# B&R Automation Studio project WithUpgradesWorking23_08_24
Automation Studio 4.9

## Configuration Config1

CPU X90CP174.48-00, AutomationRuntime I4.93, Build 4.1.2, Safety 0.0, Vc V4.72.6

### Hardware
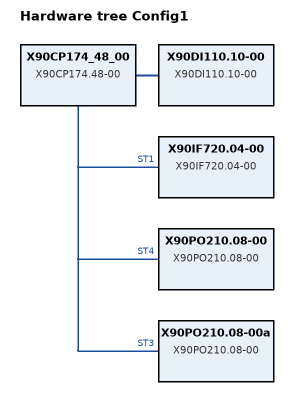
```
X90CP174_48_00 : X90CP174.48-00 v1.4.5.0  [X1 -> X1.SL]
  Module X1 (Type=X1, Virtual=true, Version=1.4.5.0)
    Connection (Connector=SL, TargetModule=X90CP174_48_00, TargetConnector=X1)
    ChannelConfig01 = 42
    DigitalFilterPin01 = 200
    ChannelConfig02 = 42
    DigitalFilterPin02 = 200
    ChannelConfig03 = 42
    DigitalFilterPin03 = 200
    ChannelConfig04 = 42
    DigitalFilterPin04 = 200
    ChannelConfig05 = 42
    DigitalFilterPin05 = 200
    ChannelConfig06 = 42
    DigitalFilterPin06 = 200
    ChannelConfig07 = 42
    DigitalFilterPin07 = 200
    ChannelConfig08 = 42
    DigitalFilterPin08 = 200
    ChannelConfig12 = 81
    ChannelConfig13 = 72
    DigitalFilterPin13 = 200
    ChannelConfig17 = 80
    ChannelConfig18 = 80
    ChannelConfig19 = 80
    ChannelConfig20 = 80
    ChannelConfig21 = 80
    ChannelConfig22 = 80
    ChannelConfig23 = 80
    IN2_InputFilter_Pin23 = 3
    ChannelConfig24 = 80
    ChannelConfig27 = 1
    ChannelConfig28 = 41
    DigitalFilterPin28 = 200
    ChannelConfig37 = 1
    LoadType37 = 2
    ChannelConfig38 = 1
    LoadType38 = 2
    ChannelConfig39 = 1
    ChannelConfig41 = 1
    LoadType41 = 2
    ChannelConfig42 = 1
    ChannelConfig45 = 1
    LoadType45 = 2
    ChannelConfig46 = 1
    LoadType46 = 2
    core = core1
  Connector IF2:
    ActivateDevice = 1
    Mode = Manual
    InternetAddress = 169.254.143.70
    SubnetMask = 255.255.0.0
    InaNodeNumber = 0
    ActivateSnmp = 2
  Connector IF3:
    DNAConfiguration = manual
    CycleTime = 1000
  ConfigurationID = Project_Config1
  UserPartitionSize = 0
  VolatileGlobalPvSize = 100000000
  IdleTaskClass = 5
  TaskClassIdleTime = 5000
  CyclicTaskClassCount = 6
  Cyclic1Duration = 1000
  Cyclic1Tolerance = 10000
  Cyclic2Duration = 4000
  Cyclic2Tolerance = 20000
  Cyclic3Duration = 10000
  Cyclic3Tolerance = 20000
  Cyclic4Duration = 20000
  Cyclic4Tolerance = 20000
  Cyclic5Duration = 50000
  Cyclic5Tolerance = 50000
  Cyclic6Duration = 100000
  Cyclic6Tolerance = 100000
  Cyclic7Duration = 100000
  Cyclic7Tolerance = 1000000
  Cyclic8Duration = 10000
  Cyclic8Tolerance = 30000000
  FileDevice1
  FileDeviceName1 = C
  FileDevicePath1 = C:/vikings/missions
  FileDevice2
  FileDeviceName2 = plc
  FileDevicePath2 = USER_PATH
  FtpUser1
  FtpUsername1 = viking  // viking
  FtpUserPassword1 = Dom8yxQRfEJkQNN0YFGST8fEunO7EPE9T/2DWtETr4U=  // viking
  FtpUserSalt1 = iKbGjPE0
  FTPAccessRight1 = 0
  ActivateOpcUa = 1
  OpcUaInformationModels_PV_Version = 1
X90DI110.10-00 : X90DI110.10-00 v1.1.1.0  [ST -> X90CP174_48_00.ST2]
  Mode_DigIn01 = 22k_pnp
  InputFilter01 = 200
  Mode_DigIn02 = 22k_pnp
  InputFilter02 = 200
  Mode_DigIn03 = 22k_pnp
  InputFilter03 = 200
  Mode_DigIn04 = 22k_pnp
  Mode_DigIn05 = 22k_pnp
  Mode_DigIn06 = 22k_pnp
  Mode_DigIn07 = 22k_pnp
  InputFilter07 = 200
  Mode_DigIn08 = 22k_pnp
  Mode_DigIn09 = 22k_pnp
  InputFilter09 = 200
  Mode_DigIn10 = 22k_pnp
  InputFilter10 = 200
X90IF720.04-00 : X90IF720.04-00 v1.0.2.0  [ST -> X90CP174_48_00.ST1]
  Connector IF4:
    Baudrate = 115200
X90PO210.08-00 : X90PO210.08-00 v1.4.0.0  [ST -> X90CP174_48_00.ST4]
X90PO210.08-00a : X90PO210.08-00 v1.4.0.0  [ST -> X90CP174_48_00.ST3]
```

### IoMap.iom - X90CP174_48_00/IoMap.iom
```iecst
VAR_CONFIG
	::gCooling.outputs.do_fan[1] AT %QX."X1".DigitalOutput46;
	::gCooling.inputs.ai_coolingTemp[0] AT %IW."X1".AnalogInput17;
	::gCooling.inputs.ai_coolingTemp[1] AT %IW."X1".AnalogInput19;
	::gCooling.outputs.do_pump[1] AT %QX."X1".DigitalOutput45;
	::gCooling.outputs.do_fan[0] AT %QX."X1".DigitalOutput37;
	::gCooling.outputs.do_pump[0] AT %QX."X1".DigitalOutput38;
	::gSafetyChain.inputs.di_interlockWheelFR_OK AT %IX."X1".DigitalInput05;
	::gSafetyChain.inputs.di_shutdownRight_OK AT %IX."X1".DigitalInput07;
	::gSafetyChain.inputs.di_interlockWheelFL_OK AT %IX."X1".DigitalInput06;
	::gSafetyChain.inputs.di_interlockWheelRR_OK AT %IX."X1".DigitalInput08;
	::gSafetyChain.inputs.di_shutdownLeft_OK AT %IX."X1".DigitalInput01;
	::gSafetyChain.inputs.di_shutdownCockpit_OK AT %IX."X1".DigitalInput02;
	::gSafetyChain.inputs.di_inertiaSwitch_OK AT %IX."X1".DigitalInput03;
	::gSafetyChain.inputs.di_BOTS_OK AT %IX."X1".DigitalInput04;
	::gSafetyChain.inputs.di_TSMS_OK AT %IX."X1".DigitalInput13;
	::gSteeringAngle.inputs.angleSensor AT %IW."X1".AnalogInput20;
	::gTorqueSensor.inputs.torque2 AT %IW."X1".AnalogInput21;
	::gBraking.inputs.ai_brakePressureFront AT %IW."X1".AnalogInput22;
	::gTorqueSensor.inputs.torque1 AT %IW."X1".AnalogInput24;
	::gBraking.inputs.ai_brakePressureRear AT %IW."X1".AnalogInput18;
	::gInverters.inverter[0].inputs.di_deratingActive AT %IX."X90DI110.10-00".DigitalInput06;
	::gInverters.inverter[1].inputs.di_deratingActive AT %IX."X90DI110.10-00".DigitalInput04;
	::gInverters.inverter[2].inputs.di_deratingActive AT %IX."X90DI110.10-00".DigitalInput08;
	::gInverters.inverter[3].inputs.di_deratingActive AT %IX."X90DI110.10-00".DigitalInput05;
	::gInverters.inverter[0].outputs.do_enable AT %QX."X90PO210.08-00a".DigitalOutput01;
	::gInverters.inverter[1].outputs.do_enable AT %QX."X90PO210.08-00a".DigitalOutput07;
	::gInverters.inverter[3].outputs.do_enable AT %QX."X90PO210.08-00a".DigitalOutput06;
	::gInverters.inverter[2].outputs.do_torqueLimitActive AT %QX."X90PO210.08-00a".DigitalOutput02;
	::gInverters.inverter[0].outputs.do_torqueLimitActive AT %QX."X90PO210.08-00a".DigitalOutput03;
	::gInverters.inverter[1].outputs.do_torqueLimitActive AT %QX."X90PO210.08-00a".DigitalOutput08;
	::gInverters.output.do_enableInv34 AT %QX."X90PO210.08-00a".DigitalOutput04;
	::gInverters.inverter[2].outputs.do_enable AT %QX."X90PO210.08-00".DigitalOutput03;
	::gInverters.inverter[3].outputs.do_torqueLimitActive AT %QX."X90PO210.08-00".DigitalOutput02;
	::gInverters.output.do_enableInv12 AT %QX."X90PO210.08-00".DigitalOutput05;
	::gSafetyChain.inputs.di_TS_Container AT %IX."X90DI110.10-00".DigitalInput07;
	::gSafetyChain.inputs.di_interlockWheelRL_OK AT %IX."X90DI110.10-00".DigitalInput10;
	::gSafetyChain.inputs.di_supply AT %IX."X90DI110.10-00".DigitalInput09;
	::gSafetyChain.inputs.di_BSPD_OK AT %IX."X90DI110.10-00".DigitalInput03;
	::gSafetyChain.inputs.di_interlockHVD_OK AT %IX."X90DI110.10-00".DigitalInput01;
	::gSafetyChain.inputs.di_interlockTSMP_OK AT %IX."X90DI110.10-00".DigitalInput02;
	::gRTDS.outputs.do_RTDS AT %QX."X1".DigitalOutput41;
	::gBraking.outputs.do_brakeLight AT %QX."X1".DigitalOutput42;
	gRTDS.inputs.im_RTDS_Current AT %IW."X1".Current41;
	::gCooling.inputs.im_pumpCurrent[1] AT %IW."X1".Current45;
	::gCooling.inputs.im_pumpCurrent[0] AT %IW."X1".Current38;
	::gInverters.output.do_powerInv12 AT %QX."X1".DigitalOutput39;
	::gInverters.output.do_powerInv34 AT %QX."X1".DigitalOutput27;
	::gLowVoltageBattery.inputs.ai_voltage AT %IW."X1".AnalogInput12;
	::gLowVoltageBattery.inputs.ai_current AT %IW."X1".AnalogInput23;
	::gSafetyChain.inputs.di_interlockMotorRL_OK AT %IX."X1".DigitalInput28;
END_VAR
```

## Logical view

Binary libraries used (declarations not repeated): operator, runtime, astime, AsIecCon, standard, AsIODiag, brsystem, asstring, ArCan, brdkUSB, AsIO, AsBrStr, sys_lib, FileIO, AsUSB, DataObj, brdkSTR, NcGlobal, MTTypes, dvframe, MpAlarmX, MpBase, MpRecipe, MpData, MTFilter 5.24.1

### Global.typ - Global data types
```iecst
TYPE
	CAN_STATES :
		(
		S_INIT,
		S_INIT_TX,
		S_INIT_RX,
		S_RUNNING,
		S_ERROR,
		S_IDLE
		);
END_TYPE
```

### Package Logical/Libraries - Global libraries

### Library Logical/Libraries/brdkSIM (ANSIC)

#### Types.typ
```iecst
TYPE
	brdkSIM_status_typ : 	STRUCT
		fbStatus : brdkSIM_STATUS_typ;
		error : BOOL;
		errorCode : UINT;
	END_STRUCT;
	brdkSIM_STATUS_typ :
		(
		brdkSIM_NOT_ENABLED := 0,
		brdkSIM_BUSY := 10,
		brdkSIM_RUNNING := 20,
		brdkSIM_ERROR := 200
		);
	brdkSimInput_internal_typ : 	STRUCT
		state : USINT;
		AsIOEnableForcing_0 : AsIOEnableForcing;
		AsIOSetForceValue_0 : AsIOSetForceValue;
		AsIODisableForcing_0 : AsIODisableForcing;
		oldSetValue : UDINT;
	END_STRUCT;
	brdkSimOutput_internal_typ : 	STRUCT
		state : USINT;
		pvStatus : UINT;
		pvAdr : UDINT;
		pvLen : UDINT;
		pvCheck : UINT;
		pvCmpString : STRING[4];
		boolVar : BOOL;
	END_STRUCT;
END_TYPE
```

#### brdkSimInput.c
```c
#include <bur/plctypes.h>
#include <AsIO.h>
#include <AsBrStr.h>

#ifdef __cplusplus
	extern "C"
	{
#endif
	#include "brdkSIM.h"
#ifdef __cplusplus
	};
#endif

#define false 0
#define true 1

/* TODO: Add your comment here */
void brdkSimInput(struct brdkSimInput* inst)
{
	int i;

	if (!inst->enable && inst->internal.state > 0 && inst->internal.state < 50) {
		inst->internal.state = 50;
	}

	switch (inst->internal.state) {
		case 0: //wait for enable force
			inst->status.fbStatus = brdkSIM_NOT_ENABLED;
			inst->status.error = false;
			inst->status.errorCode = 0;
			inst->internal.oldSetValue = 0;
			if (inst->enable) {
				inst->internal.state = 10;
			}
			break;

		case 10: //enable force
			inst->status.fbStatus = brdkSIM_BUSY;
			if (!inst->internal.AsIOEnableForcing_0.enable) {
				inst->internal.AsIOEnableForcing_0.enable = true;
				inst->internal.AsIOEnableForcing_0.pDatapoint = (UDINT)&inst->dpName;		// set pointer to the var name (address)
				inst->internal.state = 20;
			}
			break;

		case 20: //wait for AsIOEnableForcing_0 fb to be ready
			if (inst->internal.AsIOEnableForcing_0.status == ERR_OK) {
				inst->internal.AsIOEnableForcing_0.enable = false;					// remember to set enable false so the fb is ready for the next dp
				AsIOEnableForcing(&inst->internal.AsIOEnableForcing_0);
				inst->internal.state = 30;
			}
			else if (inst->internal.AsIOEnableForcing_0.status != ERR_OK && inst->internal.AsIOEnableForcing_0.status != ERR_FUB_BUSY && inst->internal.AsIOEnableForcing_0.status != ERR_FUB_ENABLE_FALSE) {
				inst->status.fbStatus = brdkSIM_ERROR;
				inst->status.error = true;
				inst->status.errorCode = inst->internal.AsIOEnableForcing_0.status;
				inst->internal.state = 200;
			}
			break;

		case 30: //AsIOSetForceValue_0 fb use to control force value
			inst->status.fbStatus = brdkSIM_RUNNING;
			inst->internal.AsIOSetForceValue_0.enable 		= true;
			inst->internal.AsIOSetForceValue_0.pDatapoint	= (UDINT)&inst->dpName;		// set pointer to the dp name (address)
			inst->internal.AsIOSetForceValue_0.value 		= inst->setValue;						// set the force value

			if (inst->internal.AsIOSetForceValue_0.status != ERR_OK && inst->internal.AsIOSetForceValue_0.status != ERR_FUB_BUSY && inst->internal.AsIOSetForceValue_0.status != ERR_FUB_ENABLE_FALSE) {
				inst->status.fbStatus = brdkSIM_ERROR;
				inst->status.error = true;
				inst->status.errorCode = inst->internal.AsIOSetForceValue_0.status;
				inst->internal.state = 200;
			}
			break;

		case 50: //set value to 0 before disable
			inst->status.fbStatus = brdkSIM_BUSY;
			if (inst->internal.AsIOSetForceValue_0.value != 0) {
				inst->internal.AsIOSetForceValue_0.enable 		= true;
				inst->internal.AsIOSetForceValue_0.pDatapoint	= (UDINT)&inst->dpName;		// set pointer to the dp name (address)
				inst->internal.AsIOSetForceValue_0.value 		= 0;									// set the force value
				inst->internal.oldSetValue 						= 0;

				if (inst->internal.AsIOSetForceValue_0.status != ERR_OK && inst->internal.AsIOSetForceValue_0.status != ERR_FUB_BUSY && inst->internal.AsIOSetForceValue_0.status != ERR_FUB_ENABLE_FALSE) {
					inst->status.fbStatus = brdkSIM_ERROR;
					inst->status.error = true;
					inst->status.errorCode = inst->internal.AsIOSetForceValue_0.status;
					inst->internal.state = 200;
				}
				else {
					inst->internal.state 	= 60;
				}
			}
			else {
				inst->internal.state 	= 60;
			}
			break;

		case 60: //wait for AsIODisableForcing_0 fb to be ready
			inst->internal.AsIOSetForceValue_0.enable 		= false;
			inst->internal.AsIODisableForcing_0.enable 		= true;
			inst->internal.AsIODisableForcing_0.pDatapoint 	= (UDINT)&inst->dpName;		// set pointer to the dp name (address)
			AsIODisableForcing(&inst->internal.AsIODisableForcing_0);

			if (inst->internal.AsIODisableForcing_0.status == ERR_OK) {
				inst->internal.AsIODisableForcing_0.enable 	= false;						// remember to set enable false so the fb is ready for the next dp
				inst->internal.state = 0;
			}
			else if (inst->internal.AsIODisableForcing_0.status != ERR_OK && inst->internal.AsIODisableForcing_0.status != ERR_FUB_BUSY && inst->internal.AsIODisableForcing_0.status != ERR_FUB_ENABLE_FALSE) {
				inst->status.fbStatus = brdkSIM_ERROR;
				inst->status.error = true;
				inst->status.errorCode = inst->internal.AsIODisableForcing_0.status;
				inst->internal.state = 200;
			}
			break;

		case 200: //error
			inst->internal.AsIOEnableForcing_0.enable = false;
			inst->internal.AsIOSetForceValue_0.enable = false;
			inst->internal.AsIODisableForcing_0.enable 	= false;
			inst->internal.oldSetValue = 0;

			if (!inst->enable) {
				inst->status.error = false;
				inst->status.errorCode = 0;
				inst->internal.state 	= 0;
			}
	}

	AsIOEnableForcing(&inst->internal.AsIOEnableForcing_0);
	AsIOSetForceValue(&inst->internal.AsIOSetForceValue_0);
	AsIODisableForcing(&inst->internal.AsIODisableForcing_0);
}
```

#### brdkSimOutput.c
```c
#include <bur/plctypes.h>
#include <sys_lib.h>
#include <AsBrStr.h>

#ifdef __cplusplus
	extern "C"
	{
#endif
	#include "brdkSIM.h"
#ifdef __cplusplus
	};
#endif

#define false 0
#define true 1

/* TODO: Add your comment here */
void brdkSimOutput(struct brdkSimOutput* inst)
{
	if (!inst->enable && inst->internal.state > 0) {
		inst->internal.state = 0;
		inst->internal.pvAdr = 0;
		inst->internal.pvCheck = 0;
		inst->internal.pvLen = 0;
		inst->internal.pvStatus = 0;
		inst->internal.state = 0;
	}

	switch (inst->internal.state) {
		case 0: //wait for enable
			inst->status.fbStatus = brdkSIM_NOT_ENABLED;
			inst->status.error = false;
			inst->status.errorCode = 0;

			if(inst->enable) {
				brsstrcpy((UDINT)inst->internal.pvCmpString, (UDINT) "");
				inst->internal.pvCheck = brsstrcmp((UDINT)inst->pvName, (UDINT)inst->internal.pvCmpString);
				if(inst->internal.pvCheck != 0) {
					inst->internal.state = 10;
				}
				else {
					inst->status.fbStatus = brdkSIM_ERROR;
					inst->status.error = true;
					inst->status.errorCode = 1000;
					inst->internal.state = 200;
				}
			}
			break;

		case 10: //get address of the pv
			inst->status.fbStatus = brdkSIM_BUSY;
			inst->internal.pvStatus = PV_xgetadr((UDINT)&inst->pvName, (UDINT)&inst->internal.pvAdr, (UDINT)&inst->internal.pvLen);

			if(inst->internal.pvStatus != 0) {
				inst->status.fbStatus = brdkSIM_ERROR;
				inst->status.error = true;
				inst->status.errorCode = inst->internal.pvStatus;
				inst->internal.state = 200;
			}
			else {
				inst->internal.state = 20;
			}
			break;

		case 20: //check value
			inst->status.fbStatus = brdkSIM_RUNNING;
			brsmemcpy((UDINT)&inst->actValue, (UDINT)inst->internal.pvAdr, inst->internal.pvLen);
			break;

		case 200: //error
			break;
	}
}
```

### Library Logical/Libraries/sduVikings (IEC)

#### calculateSensorNetOut.st
```iecst
(* TODO: Add your comment here *)
FUNCTION_BLOCK calculateSensorNetOut
//	y = a1 + a2*x^1 + a3*x^2 + a4*x^3 + ... + a8*x^7
	y := polyCoeffs[0];
	FOR i := 1 TO 8 DO
		// y = y + a^i
		y := y + polyCoeffs[i] * EXPT(INT_TO_REAL(input), i);
	END_FOR;
	output := y;
END_FUNCTION_BLOCK
```

### globalEventLog.typ - Global data types
```iecst
TYPE
	gEventLog_typ : 	STRUCT
		newEventString : STRING[80];
		logNewEvent : BOOL;
		eventIndex : UINT := 0;
		events : ARRAY[0..EVENT_LOG_LENGTH]OF STRING[80];
		resetEventLog : BOOL;
	END_STRUCT;
END_TYPE
```

### globalEventLog.var - Global variables
```iecst
VAR CONSTANT
	EVENT_LOG_LENGTH : UINT := 100;
END_VAR
VAR
	gEventLog : gEventLog_typ;
END_VAR
```

### globalStateMachine.typ
```iecst
TYPE
	gStateMachine_cmd_typ : 	STRUCT
		forceIO : BOOL;
		changeMission : BOOL;
		loadMission : BOOL;
		saveMission : BOOL;
	END_STRUCT;
	gStateMachine_data_typ : 	STRUCT
		dummy : USINT;
	END_STRUCT;
	gStateMachine_inputs_typ : 	STRUCT
		dummy : INT;
	END_STRUCT;
	gStateMachine_outputs_typ : 	STRUCT
		dummy : USINT;
	END_STRUCT;
	gStateMachine_status_typ : 	STRUCT
		readyForStateDrive : BOOL;
		stateNameOld : STRING[80];
		stateName : STRING[80];
		stateChangeAllowed : BOOL;
		stateOld : states_typ;
		state : states_typ;
		instruction : STRING[80];
		instructionIndex : instructionIndex;
		mission : STRING[80];
		missionIndex : missionIndex_typ;
		stateChangeTimeout : BOOL;
	END_STRUCT;
	gStateMachine_typ : 	STRUCT
		status : gStateMachine_status_typ;
		outputs : gStateMachine_outputs_typ;
		data : gStateMachine_data_typ;
		cmd : gStateMachine_cmd_typ;
		inputs : gStateMachine_inputs_typ;
	END_STRUCT;
	instructionIndex :
		(
		INST_INITIALIZING,
		INST_PRESS_SAFETY_BUTTON,
		INST_SC_NOT_ENABLED,
		INST_PRESS_TRACTIVE_BUTTON,
		INST_AMS_NOT_READY,
		INST_PRESS_BRAKE,
		INST_TORQUE_PEDAL_FAULT,
		INST_PRE_CHARGING,
		INST_PRESS_DRIVE_BUTTON,
		INST_FIX_ERROR,
		INST_CLOSE_SAFETY_CHAIN,
		INST_IN_DRIVE
		);
	states_typ :
		(
		STATE_INITIALIZE,
		STATE_IDLE,
		STATE_ENABLING_SC,
		STATE_SC_ENABLED,
		STATE_PRECHARGING,
		STATE_TRACTIVE,
		STATE_DRIVE,
		STATE_ERROR
		);
END_TYPE
```

### globalStateMachine.var
```iecst
VAR
	gStateMachine : gStateMachine_typ;
END_VAR
```

### Program Logical/SM/StateMachine (IEC)

#### Types.typ - Local data types
```iecst
TYPE
	this_typ : 	STRUCT
		TON_initialization : TON;
		instructionList : ARRAY[0..25]OF STRING[80];
	END_STRUCT;
END_TYPE
```

#### stateInit.st
```iecst
(* State Initialize *)
ACTION stateInit:

	this.TON_initialization();

	(* Start timer *)
	IF NOT this.TON_initialization.IN THEN
		this.TON_initialization.IN := TRUE;
	END_IF

END_ACTION

(* Conditions for state change for STATE_INITIALIZE*)
ACTION stateChangeInit:

	(* Initialization done change state to ready *)
	IF this.TON_initialization.Q THEN
		this.TON_initialization.IN := FALSE;
		gStateMachine.status.state := STATE_IDLE;
	END_IF

END_ACTION
```

#### stateEnablingSC.st
```iecst
(* State Ready *)
ACTION stateEnablingSC:
	(* Update instruction string *)
	gStateMachine.status.instructionIndex := INST_SC_NOT_ENABLED;
END_ACTION

(* Conditions for state change for STATE_ENABLE_SAFETY_CHAIN *)
ACTION stateChangeEnablingSC:
	IF gStateMachine.status.stateChangeAllowed THEN
		(* If message received from AMS saying that SC is enabled *)
		IF gAMS.status.scEnabled THEN
			gStateMachine.status.state := STATE_SC_ENABLED;
		END_IF

		(* If safety chain is broken go to state 'stateError' *)
		IF NOT gSafetyChain.status.scOK_notEnabled THEN
			gStateMachine.status.state 	:= STATE_ERROR;
			gAMS.cmd.abort 				:= TRUE;
		END_IF

		IF gStateMachine.status.stateChangeTimeout THEN
			gAMS.cmd.abort := TRUE;
			gStateMachine.status.state 			    := STATE_IDLE;
		END_IF;
	END_IF;

END_ACTION
```

#### logEvent.st
```iecst
ACTION logEvent:

	gEventLog.events[gEventLog.eventIndex] := gEventLog.newEventString;

	gEventLog.eventIndex 				   := gEventLog.eventIndex + 1;
	IF gEventLog.eventIndex > EVENT_LOG_LENGTH THEN
		gEventLog.eventIndex := 0;
	END_IF;

	gEventLog.events[gEventLog.eventIndex] := '';

END_ACTION

ACTION resetEventLog:

	FOR gEventLog.eventIndex := 0 TO EVENT_LOG_LENGTH DO
		gEventLog.events[gEventLog.eventIndex] := '';
	END_FOR;
	gEventLog.eventIndex := 0;

END_ACTION
```

#### forceIO.st
```iecst
ACTION initForceIO:
	brdkSimInput_0[0].dpName  := '%IX.X1.DigitalInput05'; 			//::gSafetyChain.inputs.di_interlockWheelFR_OK
	brdkSimInput_0[1].dpName  := '%IX.X1.DigitalInput07'; 			//:gSafetyChain.inputs.di_shutdownRight_OK
	brdkSimInput_0[2].dpName  := '%IX.X1.DigitalInput06'; 			//::gSafetyChain.inputs.di_interlockWheelFL_OK
	brdkSimInput_0[3].dpName  := '%IX.X1.DigitalInput08'; 			//::gSafetyChain.inputs.di_interlockWheelRR_OK
	brdkSimInput_0[4].dpName  := '%IX.X1.DigitalInput01'; 			//::gSafetyChain.inputs.di_shutdownLeft_OK
	brdkSimInput_0[5].dpName  := '%IX.X1.DigitalInput02'; 			//::gSafetyChain.inputs.di_shutdownCockpit_OK
	brdkSimInput_0[6].dpName  := '%IX.X1.DigitalInput03'; 			//::gSafetyChain.inputs.di_inertiaSwitch_OK
	brdkSimInput_0[7].dpName  := '%IX.X1.DigitalInput04'; 			//::gSafetyChain.inputs.di_BOTS_OK
	brdkSimInput_0[8].dpName  := '%IX.X1.DigitalInput13'; 			//::gSafetyChain.inputs.di_TSMS_OK
	brdkSimInput_0[9].dpName  := '%IW.X1.AnalogInput20'; 			//::gSteeringAngle.inputs.angleSensor
	brdkSimInput_0[10].dpName := '%IW.X1.AnalogInput21'; 			//::gTorqueSensor.inputs.torque2
	brdkSimInput_0[11].dpName := '%IW.X1.AnalogInput22'; 			//::gBraking.inputs.ai_brakePressureFront
	brdkSimInput_0[12].dpName := '%IW.X1.AnalogInput24'; 			//::gTorqueSensor.inputs.torque1
	brdkSimInput_0[13].dpName := '%IW.X1.AnalogInput18'; 			//::gBraking.inputs.ai_brakePressureRear
	brdkSimInput_0[14].dpName := '%IX.IF6.ST2.DigitalInput07'; //::gSafetyChain.inputs.di_TS_Container
	brdkSimInput_0[15].dpName := '%IX.IF6.ST2.DigitalInput10'; //::gSafetyChain.inputs.di_interlockWheelRL_OK
	brdkSimInput_0[16].dpName := '%IX.IF6.ST2.DigitalInput09'; //::gSafetyChain.inputs.di_supply
	brdkSimInput_0[17].dpName := '%IX.IF6.ST2.DigitalInput03'; //::gSafetyChain.inputs.di_BSPD_OK
	brdkSimInput_0[18].dpName := '%IX.IF6.ST2.DigitalInput01'; //::gSafetyChain.inputs.di_interlockHVD_OK
	brdkSimInput_0[19].dpName := '%IX.IF6.ST2.DigitalInput02'; //::gSafetyChain.inputs.di_interlockTSMP_OK
END_ACTION

ACTION forceIO:

	FOR i := 0 TO SIM_INPUTS-1 DO
		brdkSimInput_0[i].enable := gStateMachine.cmd.forceIO;
	END_FOR;

	brdkSimInput_0[0].setValue  := gSafetyChain.cmd.di_interlockWheelFR_OK;
	brdkSimInput_0[1].setValue  := gSafetyChain.cmd.di_shutdownRight_OK;
	brdkSimInput_0[2].setValue  := gSafetyChain.cmd.di_interlockWheelFL_OK;
	brdkSimInput_0[3].setValue  := gSafetyChain.cmd.di_interlockWheelRR_OK;
	brdkSimInput_0[4].setValue  := gSafetyChain.cmd.di_shutdownLeft_OK;
	brdkSimInput_0[5].setValue  := gSafetyChain.cmd.di_shutdownCockpit_OK;
	brdkSimInput_0[6].setValue  := gSafetyChain.cmd.di_inertiaSwitch_OK;
	brdkSimInput_0[7].setValue  := gSafetyChain.cmd.di_BOTS_OK;
	brdkSimInput_0[8].setValue  := gSafetyChain.cmd.di_TSMS_OK;
	brdkSimInput_0[9].setValue  := gSteeringAngle.cmd.angleSensor;
	brdkSimInput_0[10].setValue := gTorqueSensor.cmd.torque2;
	brdkSimInput_0[11].setValue := gBraking.cmd.brakePressureFront;
	brdkSimInput_0[12].setValue := gTorqueSensor.cmd.torque1;
	brdkSimInput_0[13].setValue := gBraking.cmd.brakePressureRear;
	brdkSimInput_0[14].setValue := gSafetyChain.cmd.di_TS_Container;
	brdkSimInput_0[15].setValue := gSafetyChain.cmd.di_interlockWheelRL_OK;
	brdkSimInput_0[16].setValue := gSafetyChain.cmd.di_supply;
	brdkSimInput_0[17].setValue := gSafetyChain.cmd.di_BSPD_OK;
	brdkSimInput_0[18].setValue := gSafetyChain.cmd.di_interlockHVD_OK;
	brdkSimInput_0[19].setValue := gSafetyChain.cmd.di_interlockTSMP_OK;

	FOR i := 0 TO SIM_INPUTS-1 DO
		brdkSimInput_0[i]();
	END_FOR;

END_ACTION
```

#### changeStateDelay.st
```iecst
//
ACTION changeStateDelay:
	IF gStateMachine.status.state <> STATE_TRACTIVE THEN
		gStateMachine.status.readyForStateDrive := FALSE;
	END_IF

	TON_stateChange(IN := gStateMachine.status.stateOld <> gStateMachine.status.state);
	IF TON_stateChange.Q THEN
		gStateMachine.status.stateOld := gStateMachine.status.state;
	END_IF;

	gStateMachine.status.stateChangeAllowed := gStateMachine.status.stateOld = gStateMachine.status.state;

END_ACTION
```

### Variables.var
```iecst
VAR
	TON_persistancetimer : TON;
	i : USINT;
END_VAR
```

### globalInverters.typ
```iecst
TYPE
	gInverters_typ : 	STRUCT
		data : gInverters_data_typ;
		cmd : gInverters_cmd_typ;
		status : gInverters_status_typ;
		output : gInverters_output_typ;
		inverter : ARRAY[0..3]OF gInverters_inverter_typ;
	END_STRUCT;
	gInverters_data_typ : 	STRUCT
		powerLimitKW : REAL;
		powerLimit : REAL;
		averageVelocityKmh : REAL;
		deratingStatic : REAL;
		acceleration_0to100kmh_inSecs : TIME;
		negativeTorqueLimGain : REAL;
		torqueSetpointGain : REAL;
		MaxSpeedRPM : REAL;
		powerLimitMargin : REAL;
		powerLimitKwInverter : ARRAY[0..3]OF REAL;
		powerBias : ARRAY[0..3]OF REAL;
		rearBias : REAL;
	END_STRUCT;
	gInverters_cmd_typ : 	STRUCT
		enableRegenerativeBraking : BOOL;
		enableTractionControl : BOOL;
		enablePowerLimiter : BOOL;
		enableTorqueVectoring : BOOL;
		enableTorqueLimiter : BOOL;
		enableFrontRearDistribution : BOOL;
		enableMotorPairShutdown : BOOL;
		powerCycle : BOOL;
		exitDrive : BOOL;
		manualControl : BOOL;
		enableConfigurationDuringDrive : BOOL; (*True = All inverter control parameters are enabled to be changed during drive*)
		autoReset : BOOL;
		stopInverters : BOOL;
		activateInverters : BOOL;
		powerCyclePair12 : BOOL;
		powerCyclePair34 : BOOL;
	END_STRUCT;
	gInverters_output_typ : 	STRUCT
		do_enableInv34 : BOOL; (*BA1*)
		do_enableInv12 : BOOL; (*BA1*)
		do_powerInv12 : BOOL;
		do_powerInv34 : BOOL;
	END_STRUCT;
	gInverters_status_typ : 	STRUCT
		deratingStaticPercent : REAL;
		configurationEnabled : BOOL;
		errorCanFramesLost : ARRAY[0..1]OF BOOL;
		regenerativeBrakingAvailable : BOOL;
		torqueBasedThrottle : BOOL;
	END_STRUCT;
	gInverters_inverter_typ : 	STRUCT
		status : gInverters_inverter_status_typ;
		outputs : gInverters_inverter_outputs_typ;
		data : gInverters_inverter_data_typ;
		inputs : gInverters_inverter_inputs_typ;
		cmd : gInverters_inverter_cmd_typ;
	END_STRUCT;
	gInverters_inverter_status_typ : 	STRUCT
		ok : BOOL;
		substate : USINT;
		stateName : STRING[80];
		state : gInverterStates;
		returnState : gInverterStates; (*State to return back to if an error occurs here*)
		errorTimeout : BOOL;
		inverterEnabled : BOOL;
		unknownMessageReceived : BOOL;
		unknownMessageID : UDINT;
		inverterDisconnected : BOOL;
		locationName : STRING[80];
		location : INVERTER_LOCATIONS_TYP;
		deratingLaunchProfilePercent : REAL;
		deratingPowerLimiterPercent : REAL;
		deratingFrontRearDistribution : REAL;
		deratingTorqueVectoringPercent : REAL;
		deratingTotalPercent : REAL;
	END_STRUCT;
	gInverters_inverter_data_typ : 	STRUCT
		torqueOutput : REAL;
		torqueOutputPercent : REAL;
		tempMotor : REAL;
		tempInverter : REAL;
		tempIGBT : REAL;
		actualVelocityKmh : REAL;
		actualVelocity : REAL;
		torqueCurrent : REAL;
		torqueMagnitizingCurrent : REAL;
		speedDerating : REAL;
		maxSpeed : REAL; (*Max speed recorded in last run, remember to implement in code*)
		TON_errorTimer : TON; (*Timer to monitor how long an inverter has been in the error state*)
		regenerativeBraking : REAL;
		regenerativeBrakingPercent : REAL;
	END_STRUCT;
	gInverters_inverter_inputs_typ : 	STRUCT
		com_systemReady : BOOL;
		com_error : BOOL;
		com_warning : BOOL;
		com_quitDcOn : BOOL;
		com_dcOn : BOOL;
		com_quitInverterOn : BOOL;
		com_inverterOn : BOOL;
		com_derating : BOOL;
		com_actualVelocity : INT;
		com_torqueCurrent : INT;
		com_magnetizingCurrent : INT;
		com_tempMotor : INT;
		com_tempInverter : INT;
		com_tempIGBT : INT;
		com_errorDiagnostics : UDINT;
		di_deratingActive : BOOL;
	END_STRUCT;
	gInverters_inverter_cmd_typ : 	STRUCT
		enableInverter : BOOL;
		stopInverter : BOOL;
		startInverter : BOOL;
		shutdownByPartner : BOOL;
		powerCycle : BOOL;
	END_STRUCT;
	gInverters_inverter_outputs_typ : 	STRUCT
		torqueEnable : BOOL;
		do_torqueLimitActive : BOOL; (*BE2*)
		do_enable : BOOL; (*BE1*)
		com_errorReset : BOOL;
		com_enable : BOOL;
		com_dcOn : BOOL;
		com_interverOn : BOOL;
		com_targetVelocity : INT;
		com_targetTorque : INT;
		com_torqueLimitPos : INT;
		com_torqueLimitNeg : INT;
	END_STRUCT;
	missionIndex_typ :
		(
		MISSION_NONE,
		MISSION_ACCELERATION,
		MISSION_SKIDPAD,
		MISSION_SPRINT,
		MISSION_ENDURANCE,
		MISSION_BRAKE_TEST,
		MISSION_TESTING
		);
	INVERTER_LOCATIONS_TYP :
		(
		FL,
		FR,
		RL,
		RR
		);
	gInverterStates :
		(
		INV_STATE_INIT,
		INV_STATE_IDLE,
		INV_STATE_SWITCH_ON,
		INV_STATE_DRIVE,
		INV_STATE_ERROR,
		INV_STATE_SWITCH_OFF,
		INV_STATE_POWER_CYCLE
		);
END_TYPE
```

### globalInverters.var
```iecst
VAR
	gInverters : {REDUND_UNREPLICABLE} gInverters_typ;
	CONVERTER_PEAK_CURRENT : REAL := 105.00;
END_VAR
VAR CONSTANT
	INVERTER_COUNT : USINT := 3;
END_VAR
```

### Program Logical/Inverters/CAN/CAN (IEC)

#### Bus.st
```iecst
ACTION Bus:

	CASE bus[i].communicationState OF
		S_INIT:
			(* PLC is not simulated. It is run on an actual PLC *)
			IF NOT gIsSimulation THEN

				(* Configure CAN port *)
				bus[i].ArCanSetBaudrate_0.DeviceName	:= bus[i].deviceName;

				bus[i].ArCanSetBaudrate_0.Execute 	:= TRUE;
				IF bus[i].ArCanSetBaudrate_0.Done THEN
					bus[i].communicationState := S_INIT_TX;
				END_IF;

				IF bus[i].ArCanSetBaudrate_0.Error THEN
					bus[i].communicationState := S_ERROR;
				END_IF;

			ELSE
				(* PLC is simulated. It is run in the simulator and no hardware is connnected *)
				bus[i].communicationState := S_IDLE;
			END_IF;
		S_INIT_TX:
			(* Configure send function block *)
			bus[i].ArCanSend_0.Enable 		:= TRUE;
			bus[i].ArCanSend_0.DeviceName 	:= bus[i].deviceName;

			IF bus[i].ArCanSend_0.Active THEN
				bus[i].communicationState := S_INIT_RX;
			END_IF;

			IF bus[i].ArCanSend_0.Error THEN
				bus[i].communicationState := S_ERROR;
			END_IF;

		S_INIT_RX:
			(* Configure receive function block *)
			bus[i].ArCanReceive_0.Enable 		:= TRUE;
			bus[i].ArCanReceive_0.DeviceName 	:= bus[i].deviceName;

			IF bus[i].ArCanReceive_0.Active THEN
				(* CAN port successfully enabled *)
				bus[i].communicationState := S_RUNNING;
			END_IF;

			IF bus[i].ArCanReceive_0.Error THEN
				bus[i].communicationState := S_ERROR;
			END_IF

		S_RUNNING:
			(* Send messages *)
			Send_Bus;

			(* Receive messages *)
			Receive_Bus;

		S_ERROR: // Error
			IF bus[i].ArCanSend_0.Error THEN
				bus[i].ArCanSend_0(Enable := FALSE);
				bus[i].ArCanSend_0(Enable := TRUE);
			END_IF;

			IF bus[i].ArCanReceive_0.Error THEN
				bus[i].ArCanReceive_0(Enable := FALSE);
				bus[i].ArCanReceive_0(Enable := TRUE);
			END_IF;

			IF bus[i].ArCanReceive_0.Error = FALSE AND bus[i].ArCanSend_0.Error = FALSE AND bus[i].ArCanSetBaudrate_0.Error = FALSE THEN
				bus[i].communicationState 	:= S_INIT;
			END_IF;
		S_IDLE: // Do nothing
	END_CASE

	IF NOT gIsSimulation THEN
		bus[i].ArCanSetBaudrate_0();
		bus[i].ArCanReceive_0();
		bus[i].ArCanSend_0();
	END_IF;

	// Service disconnection timers
	serviceDisconnectionDetection;

END_ACTION
```

#### receiveMsgs.st
```iecst
(* Inverter 1, Actual value 1 *)
ACTION Inv_ActualValue1:

	gInverters.inverter[inverterId].inputs.com_systemReady 			:= bus[i].ArCanReceive_0.ReceivedFrame.Data[1].0;
	gInverters.inverter[inverterId].inputs.com_error 				:= bus[i].ArCanReceive_0.ReceivedFrame.Data[1].1;
	gInverters.inverter[inverterId].inputs.com_warning 				:= bus[i].ArCanReceive_0.ReceivedFrame.Data[1].2;
	gInverters.inverter[inverterId].inputs.com_quitDcOn 			:= bus[i].ArCanReceive_0.ReceivedFrame.Data[1].3;
	gInverters.inverter[inverterId].inputs.com_dcOn 				:= bus[i].ArCanReceive_0.ReceivedFrame.Data[1].4;
	gInverters.inverter[inverterId].inputs.com_quitInverterOn		:= bus[i].ArCanReceive_0.ReceivedFrame.Data[1].5;
	gInverters.inverter[inverterId].inputs.com_inverterOn 			:= bus[i].ArCanReceive_0.ReceivedFrame.Data[1].6;
	gInverters.inverter[inverterId].inputs.com_derating 			:= bus[i].ArCanReceive_0.ReceivedFrame.Data[1].7;

	memcpy(ADR(gInverters.inverter[inverterId].inputs.com_actualVelocity), 		ADR(bus[i].ArCanReceive_0.ReceivedFrame.Data[2]), 2);
	memcpy(ADR(gInverters.inverter[inverterId].inputs.com_torqueCurrent), 	  	ADR(bus[i].ArCanReceive_0.ReceivedFrame.Data[4]), 2);
	memcpy(ADR(gInverters.inverter[inverterId].inputs.com_magnetizingCurrent), 	ADR(bus[i].ArCanReceive_0.ReceivedFrame.Data[6]), 2);

END_ACTION

(* Inverter 1, Actual value 2 *)
ACTION Inv_ActualValue2:
	memcpy(ADR(gInverters.inverter[inverterId].inputs.com_tempMotor), 			ADR(bus[i].ArCanReceive_0.ReceivedFrame.Data[0]), 2);
	memcpy(ADR(gInverters.inverter[inverterId].inputs.com_tempInverter), 		ADR(bus[i].ArCanReceive_0.ReceivedFrame.Data[2]), 2);
	memcpy(ADR(gInverters.inverter[inverterId].inputs.com_errorDiagnostics),	ADR(bus[i].ArCanReceive_0.ReceivedFrame.Data[4]), 2);
	memcpy(ADR(gInverters.inverter[inverterId].inputs.com_tempIGBT),  			ADR(bus[i].ArCanReceive_0.ReceivedFrame.Data[6]), 2);
END_ACTION
```

#### Send_Bus.st
```iecst
ACTION Send_Bus:

	(* Set timer *)
	bus[i].TON_sendTimer.PT := T#30ms;

	(* If timer runs out *)
	IF bus[i].TON_sendTimer.Q THEN
		// Make sure there is free spots in the TX message buffer
		IF bus[i].ArCanSend_0.NumberOfFreeBuffers > 1010 THEN
			(* Go through each message. Encode and send them *)
			FOR j := 2*i TO (2*i)+1 DO
				(* Set ID of message *)
				bus[i].sendMessages := bus[i].sendMessages + 1;
				CASE j OF
					0: bus[i].ArCanSend_0.Frame.ID := TX_CAN_ID_BASE + 16#084;
					1: bus[i].ArCanSend_0.Frame.ID := TX_CAN_ID_BASE + 16#085;
					2: bus[i].ArCanSend_0.Frame.ID := TX_CAN_ID_BASE + 16#088;
					3: bus[i].ArCanSend_0.Frame.ID := TX_CAN_ID_BASE + 16#089;
					ELSE
				END_CASE
				IF bus[i].ArCanSend_0.Frame.ID <> 0 THEN
					encodeAndSendMessage; // Encode and send message
				END_IF;
			END_FOR;
		END_IF;

		(* Reset timer *)
		bus[i].TON_sendTimer(IN:=FALSE);
	END_IF

	(* Start timer *)
	bus[i].TON_sendTimer(IN:=TRUE);

END_ACTION
```

### Program Logical/Inverters/Control/Control (IEC)

#### Main.st - Init, cyclic, exit code
```iecst
PROGRAM _INIT

	// Initialize inverter locations
	gInverters.inverter[FL].status.location 	:= FL;
	gInverters.inverter[FR].status.location 	:= FR;
	gInverters.inverter[RL].status.location 	:= RL;
	gInverters.inverter[RR].status.location 	:= RR;

	FOR i := 0 TO INVERTER_COUNT DO
		// Initialize inverter location names
		CASE gInverters.inverter[i].status.location OF
			FL: gInverters.inverter[i].status.locationName := 'FL';
			FR: gInverters.inverter[i].status.locationName := 'FR';
			RL: gInverters.inverter[i].status.locationName := 'RL';
			RR: gInverters.inverter[i].status.locationName := 'RR';
		END_CASE

		// Enable All Inverters
		gInverters.inverter[i].cmd.enableInverter 			:= TRUE;

		// Initialize the error timeout to false
		gInverters.inverter[i].status.errorTimeout 			:= FALSE;

		// Initialize the shutdown by partner feature to false
		gInverters.inverter[i].cmd.shutdownByPartner 			:= FALSE;

		(* Set default output signals *)
//		gInverters.inverter[i].outputs.do_enable 				:= TRUE;
//		gInverters.inverter[i].outputs.do_torqueLimitActive   := TRUE;

		// Set max velocity
		gInverters.inverter[i].outputs.com_targetVelocity 	:= 17000;
		// Initialize the torque output and limits to 0
		gInverters.inverter[i].outputs.com_targetTorque	 	:= 0;
		gInverters.inverter[i].outputs.com_torqueLimitNeg 	:= 0;
		gInverters.inverter[i].outputs.com_torqueLimitPos 	:= 0;

	END_FOR;

	// Torque Gain used to convert torque outputs in range [0,1] to torque in range [0,torqueSetpointGain] required by the inverters
	gInverters.data.torqueSetpointGain 		:= 2143; //constant.MAX_TORQUE * 1000/constant.NOMINAL_TORQUE ; //[0.1%] of nominal torque

	// Initialize the inverter group hardware enable signals
	gInverters.output.do_enableInv12 			:= FALSE;
	gInverters.output.do_enableInv34 			:= FALSE;

	(* Control Initialization *)

	// Intialize controller enable signals. All are initialized to OFF because the actual state is handled by the mission feature
	gInverters.cmd.enablePowerLimiter 			:= FALSE;
	gInverters.cmd.enableRegenerativeBraking 	:= FALSE;
	gInverters.cmd.enableTorqueVectoring 		:= FALSE;
	gInverters.cmd.enableTractionControl 		:= FALSE;
	gInverters.cmd.enableTorqueLimiter			:= FALSE;
	gInverters.cmd.enableFrontRearDistribution 	:= FALSE;
	gInverters.cmd.enableMotorPairShutdown 		:= FALSE;

	// Torque Vectoring
	torqueVectoringInit;

	// Traction Control
	tractionControlInit;

	// Power Limiter
	powerLimiterInit;

	// Torque Limiter
	torqueLimiterInit;

	// Regenerative Braking, RB
	regenerativeBrakingInit;

	// Front/Rear Distribution
//	frontRearDistributionInit;

	// Get cycle time
	RTInfo_0(enable := TRUE);
	cycletime := RTInfo_0.cycle_time / 1000; //[ms]

	// TEMP
	tempActivateOutputTorque := TRUE;

	gInverters.data.rearBias := 0.6;
	individualInverterTorqueEnabled := TRUE;

END_PROGRAM

PROGRAM _CYCLIC

	// Convert the speed from RPM to KMH
	convertToKmh;

	// Measure how fast the vehicle went from 0-100kmh
	accelerationMeasurement;

	// Torque off and pair control
	torqueOff;

	// Static Front Rear Distribution
//	frontRearDistributionCyclic;

	// Calculate average velocity
	gInverters.data.averageVelocityKmh := (gInverters.inverter[0].data.actualVelocityKmh + gInverters.inverter[1].data.actualVelocityKmh + gInverters.inverter[2].data.actualVelocityKmh + gInverters.inverter[3].data.actualVelocityKmh)/4.0;

	(* Run vehicle dynamic controllers *)
	// Torque vectoring
	torqueLimiterCyclic;

	// Traction Control
	tractionControlCyclic;

	// Torque Limiter
	torqueLimiterCyclic;

	// Regenerative Braking
	regenerativeBrakingCyclic;

	// Front Rear Distribution
	frontRearDistributionCyclic;

	(* Output torque *)
	FOR i := 0 TO INVERTER_COUNT DO
		gInverters.inverter[i].status.inverterEnabled := gInverters.inverter[i].cmd.enableInverter;

		// Find total output torque. [0,1], with unit [%/100]
//		gInverter[i].data.torqueOutput 	:= 	control.TC.derating_output[i] * // Traction Control, TC
//											control.PL.derating_output[i] * // Power Limiting,   PL
//											control.TL.derating_output[i];  // Torque Limiting,  TL

		// TEMP
		gInverters.inverter[i].data.torqueOutput := gTorqueSensor.status.torquePercentage/100.0;

		// Find total output torque in percent [0,100]. Only used for liveview
		gInverters.inverter[i].data.torqueOutputPercent 	:= gInverters.inverter[i].data.torqueOutput * 100.0;

		(* If inverter is enabled and in 'drive' calculate the torque output in range [0, torqueSetpointGain] *)
		IF gInverters.inverter[i].status.state = INV_STATE_DRIVE AND gInverters.inverter[i].status.inverterEnabled THEN
			torqueSetpoint[i] := gInverters.data.torqueSetpointGain * gInverters.inverter[i].data.torqueOutput;
		ELSE
			torqueSetpoint[i] := 0;
		END_IF;

		// Convert the torque setpoint to an int value
		IF gInverters.inverter[i].status.state = INV_STATE_DRIVE THEN
			IF tempActivateOutputTorque THEN
				// Calculating the target torque based on Throttle Position
				gInverters.inverter[i].outputs.com_targetTorque 	:= REAL_TO_INT(gTorqueSensor.status.torquePercentage/100 * gInverters.data.torqueSetpointGain * 4 * gInverters.data.powerBias[i] );

				// Power Limiter
				IF individualInverterTorqueEnabled THEN
					gInverters.data.powerLimitKwInverter[i] := MIN(gInverters.data.powerLimitKW,gORION.data.DCL_KW) * gInverters.data.powerBias[i];
//					gInverters.data.powerLimitKwInverter[1] := MIN(gInverters.data.powerLimitKW,gORION.data.DCL_KW) * 1 - gInverters.data.rearBias;
//					gInverters.data.powerLimitKwInverter[2] := MIN(gInverters.data.powerLimitKW,gORION.data.DCL_KW) * gInverters.data.rearBias;
//					gInverters.data.powerLimitKwInverter[3] := MIN(gInverters.data.powerLimitKW,gORION.data.DCL_KW) * gInverters.data.rearBias;
					powerLimiterCyclicIndividual;
				ELSE
					powerLimiterCyclic;
				END_IF;
				IF gInverters.status.torqueBasedThrottle THEN
	  				gInverters.inverter[i].outputs.com_torqueLimitPos := MIN(gInverters.inverter[i].outputs.com_torqueLimitPos, gInverters.inverter[i].outputs.com_targetTorque);
				END_IF;
				IF NOT gTorqueSensor.status.torqueEnabled THEN
					gInverters.inverter[i].outputs.com_torqueLimitPos 	:= 0;
					gInverters.inverter[i].outputs.com_targetTorque 	:= 0;
				END_IF;

			ELSIF tempManualControl THEN
				// Manually controlled
			ELSE
				gInverters.inverter[i].outputs.com_targetTorque := 0;
			END_IF;
		ELSE
			gInverters.inverter[i].outputs.com_targetTorque := 0;
		END_IF;

//		gInverters.inverter[i].outputs.com_targetTorque := 0;

		// Regenerative Braking
		// Get negative torque limit in range [0,1]
		gInverters.inverter[i].data.regenerativeBraking 	:= 	control.RB.negative_torque_limit[i];

		// Convert to percent [0, 100] for liveview
		gInverters.inverter[i].data.regenerativeBraking 	:= 	control.RB.negative_torque_limit[i] * 100.0;

		IF gInverters.inverter[i].status.state = INV_STATE_DRIVE AND gInverters.inverter[i].status.inverterEnabled THEN
			// If the inverter is in a state where the negative torque limit is allowed to be changed
			// calculate the torque limit by scaling the regenerative braking [0,1] by negativeTorqueLimGain to get it in
			// the range [0, negativeTorqueLimGain] required by the inverter
			//gInverters.inverter[i].outputs.com_torqueLimitNeg := REAL_TO_INT(gInverters.data.negativeTorqueLimGain * gInverters.inverter[i].data.regenerativeBraking);
		ELSE
			// If inverter is in an invalid state for controlling the negative torque limit set it to 0 which is a save value
			//gInverters.inverter[i].outputs.com_torqueLimitNeg := 0;
		END_IF;

	END_FOR;

//	history;
END_PROGRAM

PROGRAM _EXIT

END_PROGRAM
```

#### Types.typ - Local data types
```iecst
TYPE
	constant_typ : 	STRUCT
		MAX_NEG_TORQUE : REAL;
		MAX_BRAKE_PRESSURE : REAL;
		MIN_BRAKE_PRESSURE : REAL;
		REGEN_DERATING_SPEED : REAL;
		MIN_REGEN_SPEED : REAL;
		MIN_REGENERATION_VOLTAGE : REAL;
		PI : REAL;
		GEAR_RATIO : REAL;
		WHEEL_RADIUS : REAL;
		STEERING_ANGLE_MAX : REAL;
		MAX_TORQUE_VECTORING_DERATING : REAL;
		LAUNCH_PROFILE_MIN_TORQUE_PERC : REAL;
		LAUNCH_PROFILE_MIN_TORQUE : REAL;
		LAUNCH_PROFILE_MIN_SPEED : REAL;
		DERATING_AT_MAX : REAL;
		DERATING_AREA_WIDTH : REAL;
		REAR_DISTRIBUTION : REAL;
		FRONT_DISTRIBUTION : REAL;
		TORQUE_CONSTANT : REAL;
		MAX_TORQUE : REAL;
		NOMINAL_TORQUE : REAL;
	END_STRUCT;
	CONTROL_STATES :
		(
		SIMPLE,
		NONE
		);
	control_typ : 	STRUCT
		TV : torqueVectoring;
		TC : tractionControl;
		PL : powerLimiter;
		LP : launchProfile;
		TL : torqueLimiter;
		RB : regenerativeBraking;
	END_STRUCT;
END_TYPE
```

#### torqueVectoring.st
```iecst
ACTION torqueVectoringInit:
	// Initialize the controller values
	control.TV.MAX_DERATING 		:= 0.50;// [%/100]
	control.TV.MAX_STEERING_ANGLE 	:= 100; // [deg]
END_ACTION

ACTION torqueVectoringCyclic:
	// Service the controller

//	control.TV.enable 			:= gInverters.cmd.enableTorqueVectoring;
//	control.TV.torque_input 	:= gTorqueSensor.status.torquePercentage/100.00; // Torque signal [0,1]
//	control.TV.steering_angle 	:= gSteeringAngle.data.angleDegrees;
//	control.TV();
END_ACTION
```

#### tractionControl.st
```iecst
ACTION tractionControlInit:
	// Initialize the controller values
	control.TC.enable 		 := gInverters.cmd.enableTractionControl;
	control.TC.LON_SLIP_REF  := 0.1;
	FOR i := 0 TO INVERTER_COUNT DO
		control.TC.I_GAIN[i] := 0;
		control.TC.P_GAIN[i] := 0;
	END_FOR;
END_ACTION

ACTION tractionControlCyclic:
	// Service the controller

	//	control.TC.enable			:= gInverters.cmd.enableTractionControl;
//	FOR i := 0 TO INVERTER_COUNT DO
//		control.TC.longitudinal_wheel_slip[i] := 0; // Calculate
//	END_FOR
//	control.TC();
END_ACTION
```

#### torqueLimiter.st
```iecst
ACTION torqueLimiterInit:
	// Initialize the controller values
	gInverters.status.deratingStaticPercent := 100;

	control.TL.max_torque 	 := 1; // [%/100]. 0.3 = 30%
END_ACTION

ACTION torqueLimiterCyclic:
	// Service the controller

	//	control.TL.enable			:= gInverters.cmd.enableStatic;
	//	control.TL.max_torque		:= gInverters.status.deratingStaticPercent / 100.00;
	//	control.TL();
END_ACTION
```

#### accelerationMeasurement.st
```iecst
ACTION accelerationMeasurement:
	TON_acceleration_0to100.PT := T#10s;

	TON_acceleration_0to100();

	IF enableAccelerationTimer THEN
		TON_acceleration_0to100(IN 		:= (gInverters.data.averageVelocityKmh >= 0.5 AND gStateMachine.status.state = STATE_DRIVE));
		enableAccelerationTimer 		:= NOT TON_acceleration_0to100.Q;

		IF gInverters.data.averageVelocityKmh >= 100.0 THEN
			gInverters.data.acceleration_0to100kmh_inSecs := TON_acceleration_0to100.ET;
			enableAccelerationTimer 	:= FALSE;
			TON_acceleration_0to100.IN 	:= FALSE;
		END_IF;
	ELSE
		IF gInverters.data.averageVelocityKmh < 0.5 THEN
			enableAccelerationTimer 	:= TRUE;
			TON_acceleration_0to100.IN 	:= FALSE;
			gInverters.data.acceleration_0to100kmh_inSecs := T#0s;
		END_IF;
	END_IF;

END_ACTION
```

#### convertToKmh.st
```iecst
ACTION convertToKmh:
	constant.GEAR_RATIO	  := 11.0118;
	constant.WHEEL_RADIUS := 0.195;
	constant.PI 		  := 3.141592;

	FOR i := 0 TO INVERTER_COUNT DO
		// Convert from RPM to KMH
		// Speed in km/h					=  (             Number of wheel rotations                ) * (       Wheel distance traveled	      ) * (m/min to km/h)
		gInverters.inverter[i].data.actualVelocityKmh := (gInverters.inverter[i].data.actualVelocity / constant.GEAR_RATIO) * (constant.WHEEL_RADIUS * 2 * constant.PI) * 0.06;
	END_FOR;

END_ACTION
```

#### frontRearDistribution.st
```iecst
ACTION frontRearDistributionInit:
//	// Static Front/Rear distribution

//	// 0.00   => No power on front, all power on rear
//	// 100.00 => Equal amount on front and rear
//	// 200.00 => All power on front, no power on rear
//	constant.FRONT_DISTRIBUTION				:= 100.0;
//
//
//	// Initialize values
//	FOR i := 0 TO INVERTER_COUNT DO
//		IF brdkStrCmp(ADR(gInverter[i].status.locationFrontBack), ADR('F')) = 0 THEN
//			gInverter[i].status.deratingFrontRearDistribution := constant.FRONT_DISTRIBUTION;
//		ELSE
//			gInverter[i].status.deratingFrontRearDistribution := 100.0 - constant.FRONT_DISTRIBUTION;
//		END_IF;
//	END_FOR;
//END_ACTION
//
//ACTION frontRearDistributionCyclic:
//	// If static front/rear distribution is enabled add the distribution to the default amount
//	IF EDGEPOS(gInverters.cmd.enableFrontRearDistribution) THEN
//		// Write default values to front/rear distribution
//		FOR i := 0 TO INVERTER_COUNT DO
//			IF brdkStrCmp(ADR(gInverter[i].status.locationFrontBack), ADR('F')) = 0 THEN
//				gInverter[i].status.deratingFrontRearDistribution := constant.FRONT_DISTRIBUTION;
//			ELSE
//				gInverter[i].status.deratingFrontRearDistribution := 200.0 - constant.FRONT_DISTRIBUTION;
//			END_IF;
//		END_FOR;
//	END_IF;
//
//	IF gInverters.cmd.enableFrontRearDistribution THEN
//		IF i <> 0 THEN	// Inverter 0 is used as the input
//			IF brdkStrCmp(ADR(gInverter[i].status.locationFrontBack), ADR('F')) = 0 THEN
//				// If inverter is in the front
//				gInverter[i].status.deratingFrontRearDistribution := gInverter[0].status.deratingFrontRearDistribution;
//			ELSE
//				// If the inverter is in the back
//				gInverter[i].status.deratingFrontRearDistribution := 200.0 - gInverter[0].status.deratingFrontRearDistribution;
//			END_IF;
//		END_IF;
//
//	ELSE
//		// Distribution disabled
//		gInverter[i].status.deratingFrontRearDistribution := 100.0;
//	END_IF
//	// Convert from range [0, 200] to range [0,2]
//	gInverter[i].data.deratingFrontRearDistribution := gInverter[i].status.deratingFrontRearDistribution / 100.0;
END_ACTION

ACTION frontRearDistributionCyclic:
	gInverters.data.powerBias[0] := (1 - gInverters.data.rearBias) / 2;
	gInverters.data.powerBias[1] := (1 - gInverters.data.rearBias) / 2;
	gInverters.data.powerBias[2] := (gInverters.data.rearBias) / 2;
	gInverters.data.powerBias[3] := (gInverters.data.rearBias) / 2;
END_ACTION
```

### Program Logical/Inverters/Inv_statemachine/Inv_statemachine (IEC)

#### Main.st - Init, cyclic, exit code
```iecst
PROGRAM _INIT
	(* Actions *)
	missionInit;

	(* Variable initializations  *)
	gInverters.cmd.autoReset := TRUE;

	(* Inverter Statuses *)
	FOR i := 0 TO INVERTER_COUNT DO
		// Determine if the inverters have errors or not
		gInverters.inverter[i].status.ok := 	NOT gInverters.inverter[i].status.inverterDisconnected AND
									gInverters.inverter[i].status.inverterEnabled AND
									(gInverters.inverter[i].status.state = INV_STATE_IDLE OR gInverters.inverter[i].status.state = INV_STATE_DRIVE OR gInverters.inverter[i].status.state = INV_STATE_SWITCH_ON);
	END_FOR;

	(* Intialize all inverter states *)
	FOR i := 0 TO INVERTER_COUNT DO
		gInverters.inverter[i].status.state  := INV_STATE_INIT;
	END_FOR;

//	gInverters.inverter[0].cmd.setModeManual := TRUE;

	TON_powerInv34.PT := T#1s;
	TON_powerInv34.IN := TRUE;

	TON_powerCycle[0].PT := T#5s;
	TON_powerCycle[1].PT := T#5s;

	gInverters.cmd.manualControl := FALSE;

	gInverters.cmd.enableConfigurationDuringDrive := FALSE;		// As default - Configuration of inverter parameters is not allowed during drive

	gInverters.output.do_enableInv12 	:= TRUE;
	gInverters.output.do_enableInv34 	:= TRUE;

	gInverters.cmd.activateInverters := FALSE;
END_PROGRAM

PROGRAM _CYCLIC

	(* Actions *)
	hmiAction;
	missionCyclic;

	gInverters.status.configurationEnabled := (gStateMachine.status.state <> STATE_DRIVE) OR gInverters.cmd.enableConfigurationDuringDrive;

	// Handle start and stop commands for the inverters depending on the car global state machine

	gInverters.cmd.activateInverters := gStateMachine.status.state = STATE_DRIVE;

//	gInverters.cmd.activateInverters := gStateMachine.status.state = STATE_DRIVE AND tempActivateInvsWhenInDrive;
	gInverters.cmd.stopInverters 	 := NOT gInverters.cmd.activateInverters;

	(* Mirror commands *)
	FOR i := 0 TO INVERTER_COUNT DO
		gInverters.inverter[i].cmd.startInverter := gInverters.cmd.activateInverters;
		gInverters.inverter[i].cmd.stopInverter  := gInverters.cmd.stopInverters;
	END_FOR;

	TON_powerInv34();

	gInverters.inverter[1].cmd.powerCycle := gInverters.inverter[0].cmd.powerCycle := gInverters.cmd.powerCyclePair12;
	gInverters.inverter[3].cmd.powerCycle := gInverters.inverter[2].cmd.powerCycle := gInverters.cmd.powerCyclePair34;

	IF gStateMachine.status.state <> STATE_INITIALIZE THEN
		FOR i := 0 TO INVERTER_COUNT DO
			CASE gInverters.inverter[i].status.state OF
				INV_STATE_INIT:
					gInverters.inverter[i].status.stateName := 'Initialization';
					gInverters.output.do_powerInv12 := TRUE;

					IF TON_powerInv34.Q OR i < 2 THEN
						IF TON_powerInv34.Q THEN
							gInverters.output.do_powerInv34 	:= TRUE;
							TON_powerInv34.IN 					:= FALSE;
						END_IF;
						gInverters.inverter[i].status.state 	:= INV_STATE_IDLE;
					END_IF

				INV_STATE_IDLE:
					gInverters.inverter[i].status.stateName := 'Idle';

					// If the start command has been send to the inverter. Start it up
					IF gInverters.inverter[i].cmd.startInverter THEN
						gInverters.inverter[i].status.state 		:= INV_STATE_SWITCH_ON;
						gInverters.inverter[i].status.substate 		:= 0;
					END_IF;

					// If an error occurs. Go to error state
					// OR NOT gInverters.inverter[i].inputs.com_systemReady
					IF gInverters.inverter[i].inputs.com_error OR (gInverters.inverter[i].status.inverterDisconnected AND NOT gIsSimulation) THEN
						gInverters.inverter[i].status.state 		:= INV_STATE_ERROR;
						gInverters.inverter[i].status.returnState 	:= INV_STATE_IDLE;
						gInverters.inverter[i].status.substate 		:= 0;
					END_IF;

				INV_STATE_SWITCH_ON:
					gInverters.inverter[i].status.stateName := 'Switching ON';
					CASE gInverters.inverter[i].status.substate OF
						0:  // System ready
							IF  gInverters.inverter[i].inputs.com_systemReady THEN;
								gInverters.inverter[i].status.substate 			:= 10;
							END_IF;

						10: // Turn on DC
	//						IF NOT gInverters.inverter[i].cmd.setModeManual THEN
								gInverters.inverter[i].outputs.com_dcOn 		:= TRUE;
	//						END_IF;
							// Change state when precharge is done
							IF  gInverters.inverter[i].inputs.com_dcOn AND gInverters.inverter[i].inputs.com_quitDcOn THEN
								gInverters.inverter[i].status.substate 			:= 20;
							END_IF;

						20: // Set torque limits
							gInverters.inverter[i].outputs.com_torqueLimitPos 	:= 0;
							gInverters.inverter[i].outputs.com_torqueLimitNeg 	:= 0;
							gInverters.inverter[i].status.substate 				:= 30;

						30: // Some hardware stuff
							// SET EF/EF2 = TRUE
							IF i = 0 OR i = 1 THEN
								gInverters.output.do_enableInv12 := TRUE;
							ELSE
								gInverters.output.do_enableInv34 := TRUE;
							END_IF;
							gInverters.inverter[i].status.substate 				:= 35;
						35:
							// X140 binary input BE1 = TRUE
							gInverters.inverter[i].outputs.do_enable          	:= TRUE;
							gInverters.inverter[i].status.substate 				:= 40;

						40: // Enable inverter
	//						IF NOT gInverters.inverter[i].cmd.setModeManual THEN
								gInverters.inverter[i].outputs.com_enable 		:= TRUE;
	//						END_IF;
							gInverters.inverter[i].status.substate 				:= 50;

						50: // Turn inverter ON
	//						IF NOT gInverters.inverter[i].cmd.setModeManual THEN
								gInverters.inverter[i].outputs.com_interverOn 	:= TRUE;
	//						END_IF;

							IF gInverters.inverter[i].inputs.com_inverterOn AND gInverters.inverter[i].inputs.com_quitInverterOn THEN
								gInverters.inverter[i].status.substate 			:= 60;
							END_IF;

						60: // More hardware stuff
							// Set X140 binary input BE2 = 1
							gInverters.inverter[i].outputs.do_torqueLimitActive := TRUE;
							gInverters.inverter[i].status.substate 		  		:= 200;

						200: // Start up complete. Go into drive
							gInverters.inverter[i].status.state 				:= INV_STATE_DRIVE;
							gInverters.inverter[i].status.substate 				:= 0;

					END_CASE;

					IF gInverters.inverter[i].cmd.stopInverter THEN
						gInverters.inverter[i].status.state 	:= INV_STATE_SWITCH_OFF;
						gInverters.inverter[i].status.substate 	:= 0;
					END_IF;

					// If an error occurs. Go to error state
					IF gInverters.inverter[i].inputs.com_error OR NOT gInverters.inverter[i].inputs.com_systemReady OR (gInverters.inverter[i].status.inverterDisconnected AND NOT gIsSimulation) THEN
						gInverters.inverter[i].status.state 		:= INV_STATE_ERROR;
						gInverters.inverter[i].status.returnState 	:= INV_STATE_SWITCH_ON;
						gInverters.inverter[i].status.substate 		:= 0;
					END_IF;

				INV_STATE_DRIVE:
					gInverters.inverter[i].status.stateName := 'Drive';

					// Check if inverter is in auto mode
	//				IF NOT gInverters.inverter[i].inputs.cmd_manual THEN
	//					gInverters.inverter[i].outputs.com_targetVelocity := 0;
	//					gInverters.inverter[i].outputs.com_torqueLimitPos := 0;
	//					gInverters.inverter[i].outputs.com_torqueLimitNeg := 0;
	//				END_IF;

					// Check if the stop commando has been send
					IF gInverters.inverter[i].cmd.stopInverter THEN
						gInverters.inverter[i].status.state 	:= INV_STATE_SWITCH_OFF;
						gInverters.inverter[i].status.substate 	:= 0;
					END_IF;

					// If an error occurs. Go to error state
					IF gInverters.inverter[i].inputs.com_error OR NOT gInverters.inverter[i].inputs.com_systemReady OR (gInverters.inverter[i].status.inverterDisconnected AND NOT gIsSimulation) THEN
						gInverters.inverter[i].status.state 			:= INV_STATE_ERROR;
						gInverters.inverter[i].status.returnState 		:= INV_STATE_SWITCH_ON;
						gInverters.inverter[i].status.substate 			:= 0;
					END_IF;

				INV_STATE_SWITCH_OFF:
					gInverters.inverter[i].status.stateName := 'Switching OFF';

					CASE gInverters.inverter[i].status.substate OF
						0: // Reset all setpoints
							gInverters.inverter[i].outputs.com_targetTorque 	:= 0;
							gInverters.inverter[i].outputs.com_torqueLimitPos 	:= 0;
							gInverters.inverter[i].outputs.com_torqueLimitNeg 	:= 0;
							gInverters.inverter[i].status.substate 				:= 10;

						10: // Hardware stuff
							// X140 binary input BE2 = FALSE
							gInverters.inverter[i].outputs.do_torqueLimitActive :=FALSE;
							gInverters.inverter[i].status.substate 			:= 20;

						20: // Turn off inverter
							gInverters.inverter[i].outputs.com_interverOn 	:= FALSE;
							gInverters.inverter[i].status.substate 			:= 30;

						30: // Disable inverter
							gInverters.inverter[i].outputs.com_enable 		:= FALSE;
							gInverters.inverter[i].status.substate 			:= 40;

						40: // Inverter turned off
							IF NOT gInverters.inverter[i].inputs.com_quitInverterOn THEN
								gInverters.inverter[i].status.substate 		:= 50;
							END_IF;

						50: // More hardware stuff
							// SET EF/EF2 = FALSE
							IF i = 0 OR i = 1 THEN
								gInverters.output.do_enableInv12 := FALSE;
							ELSE
								gInverters.output.do_enableInv34 := FALSE;
							END_IF;
							gInverters.inverter[i].status.substate 			:= 55;
						55:
							// X140 binary input BE1 = FALSE
							gInverters.inverter[i].outputs.do_enable        := FALSE;
							gInverters.inverter[i].status.substate 			:= 60;

						60: // Turn DC OFF
							gInverters.inverter[i].outputs.com_dcOn 		:= FALSE;
							gInverters.inverter[i].status.substate 			:= 70;

						70: // Check that DC is off
							IF NOT gInverters.inverter[i].inputs.com_quitDcOn THEN
								gInverters.inverter[i].status.substate 		:= 80;
							END_IF;
							gInverters.inverter[i].status.substate 			:= 200;

						200: // Change state
							gInverters.inverter[i].status.state 			:= INV_STATE_IDLE;
							gInverters.inverter[i].status.substate 			:= 0;

					END_CASE;

					// If an error occurs. Go to error state
					IF gInverters.inverter[i].inputs.com_error OR NOT gInverters.inverter[i].inputs.com_systemReady OR (gInverters.inverter[i].status.inverterDisconnected AND NOT gIsSimulation) THEN
						gInverters.inverter[i].status.state 				:= INV_STATE_ERROR;
						gInverters.inverter[i].status.returnState 			:= INV_STATE_IDLE;
						gInverters.inverter[i].status.substate 				:= 0;
					END_IF;

				// Error state - Hard error. System needs to be reset in some way
				INV_STATE_ERROR:
					gInverters.inverter[i].status.stateName := 'Error';
					IF NOT gInverters.cmd.manualControl THEN
						CASE gInverters.inverter[i].status.substate OF

							// Turn drive off
							0: // Reset all setpoints
								gInverters.inverter[i].outputs.com_torqueLimitNeg 	:= 0;
								gInverters.inverter[i].outputs.com_torqueLimitPos 	:= 0;
								gInverters.inverter[i].outputs.com_targetTorque   	:= 0;

								gInverters.inverter[i].status.substate 				:= 10;
							10: // Turn off inverter
								gInverters.inverter[i].outputs.com_interverOn 		:= FALSE;
								gInverters.inverter[i].status.substate 				:= 20;

							20: // Set enable to false
								gInverters.inverter[i].outputs.com_enable 			:= FALSE;
								gInverters.inverter[i].status.substate 				:= 30;

							30: // Turn off torque
								// DI2 = 0
								gInverters.inverter[i].status.substate 				:= 40;

							40: // Turn off control
								// DI1 = 0
								gInverters.inverter[i].outputs.do_enable 			:= FALSE;
								gInverters.inverter[i].outputs.do_torqueLimitActive := FALSE;
	//							IF i = 0 OR i = 1 THEN
	//								gInverters.output.do_enableInv12 				:= FALSE;
	//							ELSE
	//								gInverters.output.do_enableInv34 				:= FALSE;
	//							END_IF;

								gInverters.inverter[i].status.substate 				:= 100;

							// Eliminate cause of error
							100:

								(*

								DO SOMETHING. ELIMINATE EVERYTHING.

								*)

								// If error is gone
								IF (NOT gInverters.inverter[i].inputs.com_error) AND (NOT gInverters.inverter[i].status.inverterDisconnected OR gIsSimulation) AND
									(NOT gInverters.cmd.manualControl) AND (gInverters.inverter[i].inputs.com_systemReady) THEN
									gInverters.inverter[i].status.substate 		:= 200;
								END_IF

							200: // Start back up
								// Return to the specified return-state
								gInverters.inverter[i].status.state 	:= gInverters.inverter[i].status.returnState;
								gInverters.inverter[i].status.substate 	:= 0;
						END_CASE;
					END_IF;

				 	// Stop button pressed. Disable everything and go to idle
					IF gInverters.inverter[i].cmd.stopInverter THEN
						// Disable everything
						gInverters.inverter[i].outputs.com_dcOn 				:= FALSE;
						gInverters.inverter[i].outputs.com_enable 				:= FALSE;
						gInverters.inverter[i].outputs.com_interverOn 			:= FALSE;
						gInverters.inverter[i].outputs.com_targetTorque 		:= 0;
						gInverters.inverter[i].outputs.com_torqueLimitNeg 		:= 0;
						gInverters.inverter[i].outputs.com_torqueLimitPos 		:= 0;
						IF NOT gInverters.cmd.manualControl THEN
							gInverters.inverter[i].outputs.do_enable 				:= FALSE;
							gInverters.inverter[i].outputs.do_torqueLimitActive 	:= FALSE;
						END_IF;

//						IF i = 0 OR i = 1 THEN
//							gInverters.output.do_enableInv12 := FALSE;
//						ELSE
//							gInverters.output.do_enableInv34 := FALSE;
//						END_IF;
	//					// Switch state
	//					gInverters.inverter[i].status.state 	:= INV_STATE_IDLE;
	//					gInverters.inverter[i].status.substate 	:= 0;
					END_IF;

				INV_STATE_POWER_CYCLE:
					gInverters.inverter[i].status.stateName := 'Power Cycling';

					IF i = 0 OR i = 1 THEN
						TON_powerCycle[0].IN := TRUE;
						gInverters.output.do_powerInv12 := FALSE;
						IF TON_powerCycle[0].Q THEN
							TON_powerCycle[0].IN := FALSE;
							gInverters.inverter[i].status.state  := INV_STATE_INIT;
						END_IF;
					ELSIF i = 2 OR i = 3 THEN
						TON_powerCycle[1].IN := TRUE;
						gInverters.output.do_powerInv34 := FALSE;
						IF TON_powerCycle[1].Q THEN
							TON_powerCycle[1].IN := FALSE;
							gInverters.inverter[i].status.state  := INV_STATE_INIT;
							TON_powerInv34.IN := TRUE;
						END_IF;
					END_IF;

					IF gInverters.inverter[i].cmd.stopInverter THEN
						gInverters.inverter[i].status.state 		:= INV_STATE_IDLE;
						gInverters.inverter[i].status.substate 	:= 0;
					END_IF;
			END_CASE;

			IF gInverters.cmd.autoReset THEN
				// Small error - Soft reset without removing the motor from 'drive'
				gInverters.inverter[i].outputs.com_errorReset := gInverters.inverter[i].inputs.com_error;
			END_IF;

			// If inverter is commanded to power cycle. Change its state to STATE_POWER_CYCLE
			IF gInverters.inverter[i].cmd.powerCycle THEN
				gInverters.inverter[i].status.state   := INV_STATE_POWER_CYCLE;
				gInverters.inverter[i].cmd.powerCycle := FALSE;
			END_IF;

			(* Control the error timeout *)
			errorTimeout;

		END_FOR;
	END_IF;

	TON_powerCycle[0]();
	TON_powerCycle[1]();

	FOR i := 0 TO INVERTER_COUNT DO
		IF gInverters.cmd.powerCycle THEN
			gInverters.inverter[i].status.state  := INV_STATE_POWER_CYCLE;
		END_IF;
	END_FOR;

	FOR i := 0 TO INVERTER_COUNT DO
//	i := 2;
		IF gInverters.inverter[i].status.stateName <> oldStateName[i] THEN
			gEventLog.newEventString := 'Inv';
			IF    i = 0 THEN strcat(ADR(gEventLog.newEventString),ADR('1 '));
			ELSIF i = 1 THEN strcat(ADR(gEventLog.newEventString),ADR('2 '));
			ELSIF i = 2 THEN strcat(ADR(gEventLog.newEventString),ADR('3 '));
			ELSE 			 strcat(ADR(gEventLog.newEventString),ADR('4 '));
			END_IF;

			strcat(ADR(gEventLog.newEventString),ADR('now in state: '));
			strcat(ADR(gEventLog.newEventString),ADR(gInverters.inverter[i].status.stateName));
			logEvent;
		END_IF;
		oldStateName[i] := gInverters.inverter[i].status.stateName;
	END_FOR;

	gInverters.cmd.stopInverters := FALSE;

END_PROGRAM

PROGRAM _EXIT
	(* Insert code here *)

END_PROGRAM
```

#### Types.typ - Local data types
```iecst
TYPE
	mission_typ : 	STRUCT
		missionList : ARRAY[0..MAX_MISSIONS]OF STRING[80];
		MpRecipeRegPar_0 : ARRAY[0..MAX_MISSION_PARAMETERS]OF MpRecipeRegPar;
		MpRecipeXml_0 : MpRecipeXml;
		missionOld : missionIndex_typ;
	END_STRUCT;
END_TYPE
```

#### Variables.var - Local variables
```iecst
VAR
	tempActivateInvsWhenInDrive : BOOL := FALSE;
	oldStateName : ARRAY[0..3] OF STRING[80];
	i : INT;
	TON_powerInv34 : TON;
	TON_powerCycle : ARRAY[0..1] OF TON;
	missions : mission_typ;
END_VAR
VAR CONSTANT
	MAX_MISSION_PARAMETERS : USINT := 10;
	MAX_MISSIONS : USINT := 6;
END_VAR
```

#### errorTimeout.st
```iecst
(* If the inverter is in the error state for too long report an error *)
ACTION errorTimeout:
	(* Disable error timer if the inverter exists error state *)
	gInverters.inverter[i].data.TON_errorTimer.PT 	:= T#10s;													// Set error timeout duration
	gInverters.inverter[i].data.TON_errorTimer.IN 	:= gInverters.inverter[i].status.state = INV_STATE_ERROR; 	// enable timer if inverter is in STATE_ERROR
	gInverters.inverter[i].data.TON_errorTimer();																// Handle timer
	gInverters.inverter[i].status.errorTimeout 		:= gInverters.inverter[i].data.TON_errorTimer.Q;			// If timer runs out trigger errorTimeout
END_ACTION
```

- logEvent.st (reference to Logical/SM/StateMachine/functions/eventLog/logEvent.st)

### Program Logical/Inverters/Simulation/Simulation

#### Main.st
```iecst
PROGRAM _INIT

	gIsSimulation 	:= DiagCpuIsSimulated();

END_PROGRAM

PROGRAM _CYCLIC
	IF gIsSimulation THEN
		FOR i := 0 TO INVERTER_COUNT DO
			CASE gInverters.inverter[i].status.state OF
				INV_STATE_IDLE:
					gInverters.inverter[i].inputs.com_systemReady 		:= TRUE;

				INV_STATE_SWITCH_ON:
					gInverters.inverter[i].inputs.com_systemReady 		:= TRUE;
					IF gInverters.inverter[i].outputs.com_dcOn THEN
						gInverters.inverter[i].inputs.com_dcOn 			:= TRUE;
						gInverters.inverter[i].inputs.com_quitDcOn 		:= TRUE;
					ELSE
						gInverters.inverter[i].inputs.com_dcOn 			:= FALSE;
						gInverters.inverter[i].inputs.com_quitDcOn 		:= FALSE;
					END_IF;

					IF gInverters.inverter[i].outputs.com_interverOn THEN
						gInverters.inverter[i].inputs.com_quitInverterOn 	:= TRUE;
					ELSE
						gInverters.inverter[i].inputs.com_quitInverterOn 	:= FALSE;
					END_IF;

				INV_STATE_DRIVE:

				INV_STATE_SWITCH_OFF:
					IF NOT gInverters.inverter[i].outputs.com_interverOn THEN
						gInverters.inverter[i].inputs.com_quitInverterOn 	:= FALSE;
					ELSE
						gInverters.inverter[i].inputs.com_quitInverterOn 	:= TRUE;
					END_IF;

					IF NOT gInverters.inverter[i].outputs.com_dcOn THEN
						gInverters.inverter[i].inputs.com_quitDcOn 		:= FALSE;
					ELSE
						gInverters.inverter[i].inputs.com_quitDcOn 		:= TRUE;
					END_IF;
				INV_STATE_ERROR:
			END_CASE;
		END_FOR;
	END_IF;

END_PROGRAM

PROGRAM _EXIT

END_PROGRAM
```

### globalAMS.typ
```iecst
TYPE
	gAMS_cmd_typ : 	STRUCT
		chargingPrescalerAmp : REAL;
		chargingPrescalerPercent : USINT;
		bankCount : USINT;
		mpo1 : USINT;
		mpo2 : USINT;
		mpo3 : USINT;
		mpe : USINT;
		commandId : USINT;
		startPrecharge : BOOL;
		enableSC : BOOL;
		enterDrive : BOOL;
		abort : BOOL;
	END_STRUCT;
	gAMS_data_history_typ : 	STRUCT
		actPower : ARRAY[0..999]OF REAL;
		actCurrent : ARRAY[0..999]OF REAL;
		actSoc : ARRAY[0..999]OF REAL;
		actVoltage : ARRAY[0..999]OF REAL;
	END_STRUCT;
	gAMS_data_typ : 	STRUCT
		stateOfCharge : REAL;
		outputCurrent : REAL;
		chargeCurrent : REAL;
		batteryVoltage : REAL;
		cellTempMax : REAL;
		cellVoltageMax : ARRAY[0..4]OF REAL;
		cellVoltageMin : ARRAY[0..4]OF REAL;
		bankTemperatureMax : ARRAY[0..4]OF REAL;
		bankTemperatureMin : ARRAY[0..4]OF REAL;
		bankResistorTemperatureMax : ARRAY[0..4]OF REAL;
		bankResistorTemperatureMin : ARRAY[0..4]OF REAL;
		history : gAMS_data_history_typ;
		packPower : REAL;
		cellVoltageMinOrion : REAL;
	END_STRUCT;
	gAMS_inputs_typ : 	STRUCT
		dummy : USINT;
	END_STRUCT;
	gAMS_outputs_typ : 	STRUCT
		com_idle : BOOL;
		com_sc_enable : BOOL;
		com_precharge : BOOL;
		com_drive : BOOL;
		com_charge : BOOL;
		com_resetShunt : BOOL;
	END_STRUCT;
	gAMS_status_bank_typ : 	STRUCT
		bankVoltage : REAL;
		resistorTemperature : ARRAY[0..13]OF REAL;
		temperatures : ARRAY[0..9]OF REAL;
		cellVoltage : ARRAY[0..27]OF REAL;
	END_STRUCT;
	gAMS_status_error_typ : 	STRUCT
		errorTimers : ARRAY[0..21]OF TON;
		amsError : BOOL;
		imdError : BOOL;
		hvdcInterlockError : BOOL;
		tempWarn : BOOL;
		voltWarn : BOOL;
		precharge : BOOL;
		airMinus : BOOL;
		airPlus : BOOL;
		lowVoltage : BOOL;
		highVoltage : BOOL;
		lowTemp : BOOL;
		highTemp : BOOL;
		ltc6813Com : BOOL;
		shuntCom : BOOL;
		openSc : BOOL;
		closeSc : BOOL;
		openAirMinus : BOOL;
		closeAirMinus : BOOL;
		openAirPlus : BOOL;
		closeAirPlus : BOOL;
		openPrePlus : BOOL;
		closePrePlus : BOOL;
		preTimeout : BOOL;
		unexpectedChargeRate : BOOL;
		bankCountMismatch : BOOL;
		unexpectedTsCurrent : BOOL;
		relayFailed : BOOL;
		scBroken : BOOL;
		unfitChargeVoltage : BOOL;
		monitorError : BOOL;
	END_STRUCT;
	gAMS_status_pack_typ : 	STRUCT
		packVoltage : REAL;
		resistorTemperature : ARRAY[0..69]OF REAL;
		temperatures : ARRAY[0..49]OF REAL;
		InstantCellVoltage : ARRAY[0..179]OF REAL;
		cellTempMax : SINT;
		cellVoltage : ARRAY[0..179]OF REAL;
	END_STRUCT;
	gAMS_status_failsafe_typ : 	STRUCT
		failsafeStatus : UINT;
	END_STRUCT;
	gAMS_status_relay_typ : 	STRUCT
		dischargeRelayEnabled : BOOL;
		chargeRelayEnabled : BOOL;
		chargerSafetyEnabled : BOOL;
		malfunctionIndicatorActive : BOOL;
		MPI1SignalStatus : BOOL;
		alwaysOnSignalStatus : BOOL;
		isReadyInputStatus : BOOL;
		isChargingInputStatus : BOOL;
		MPI2SignalStatus : BOOL;
		MPI3SignalStatus : BOOL;
		chargeModeStatus : BOOL;
		MPO2SignalStatus : BOOL;
		MPO3SignalStatus : BOOL;
		MPO4SignalStatus : BOOL;
		MPEnableSignalStatus : BOOL;
		MPO1SignalStatus : BOOL;
		relayState : UINT;
	END_STRUCT;
	gAMS_status_typ : 	STRUCT
		ok : BOOL;
		pack : gAMS_status_pack_typ;
		bank : ARRAY[0..4]OF gAMS_status_bank_typ;
		error : gAMS_status_error_typ;
		hasError : BOOL;
		amsBankCount : USINT;
		amsStateName : STRING[80];
		amsState : USINT;
		amsTurnedOnCharger : BOOL;
		scEnabled : BOOL;
		highPowerWarning : BOOL;
		highPowerError : BOOL;
		disconnected : BOOL;
		prechargingDone : BOOL;
		Counter : USINT;
		relayState : gAMS_status_relay_typ;
		failsafeStatus : gAMS_status_failsafe_typ;
		DTC1Status : UINT;
		DTC2Status : UINT;
		RelayError : USINT;
		errorInfo : STRING[80];
	END_STRUCT;
	gAMS_typ : 	STRUCT
		status : gAMS_status_typ;
		outputs : gAMS_outputs_typ;
		data : gAMS_data_typ;
		inputs : gAMS_inputs_typ;
		cmd : gAMS_cmd_typ;
	END_STRUCT;
END_TYPE
```

### globalShunt.typ
```iecst
TYPE
	gShunt_typ : 	STRUCT
		data : gShunt_data_typ;
		status : gShunt_status_typ;
	END_STRUCT;
	gShunt_data_typ : 	STRUCT
		currentThreshold : REAL;
		actCurrent : REAL;
		actVoltage : REAL;
		actVoltage2 : REAL;
		actPowerKW : REAL;
		actPowerW : REAL;
		actCurrentAS : REAL;
		actPowerKWH : REAL;
		actPowerWH : REAL;
		actTemp : REAL;
	END_STRUCT;
	gShunt_status_typ : 	STRUCT
		ok : BOOL;
		disconnected : BOOL;
		currentRunning : BOOL;
	END_STRUCT;
END_TYPE
```

### globalAMS.var
```iecst
VAR
	gAMS : gAMS_typ;
END_VAR
VAR CONSTANT
	RESISTOR_COUNT : USINT := 14;
	TEMPERATURE_COUNT : USINT := 10;
	CELL_COUNT : USINT := 28;
	BANK_COUNT : USINT := 4;
	AMS_STATE_NONE : USINT := 0;
	AMS_STATE_INIT : USINT := 1;
	AMS_STATE_IDLE : USINT := 2;
	AMS_STATE_ERROR : USINT := 4;
	AMS_STATE_SC_ENABLED : USINT := 5;
	AMS_STATE_TC_ENABLED : USINT := 11;
	AMS_STATE_DRIVE : USINT := 12;
	prechargeResistance : REAL := 1000;
	requiredPrechargeLevel : REAL := 0.96;
END_VAR
VAR
	prechargeLevelReached : BOOL;
END_VAR
```

### Program Logical/AMS_and_Shunt/AMS (IEC)

#### Types.typ - Local data types
```iecst
TYPE
	constant_typ : 	STRUCT
		fullBatteryCapacitykWh : REAL;
		fullBatteryCapacityAh : REAL;
		chargingCurrentMax : REAL;
	END_STRUCT;
END_TYPE
```

#### history.st
```iecst
ACTION history:

	// Power history
	TON_historyPower.PT := powerHistoryInverval;
	TON_historyPower.IN := TRUE;
	IF TON_historyPower.Q THEN
		FOR i := 999 TO 1 BY -1 DO
			gAMS.data.history.actPower[i] := gAMS.data.history.actPower[i-1];
		END_FOR;
		gAMS.data.history.actPower[0] := gShunt.data.actPowerKW;
		TON_historyPower.IN := FALSE;
	END_IF;
	TON_historyPower();

	// Current history
	TON_historyCurrent.PT := currentHistoryInverval;
	TON_historyCurrent.IN := TRUE;
	IF TON_historyCurrent.Q THEN
		FOR i := 999 TO 1 BY -1 DO
			gAMS.data.history.actCurrent[i] := gAMS.data.history.actCurrent[i-1];
		END_FOR;
		gAMS.data.history.actCurrent[0] := gShunt.data.actCurrent;
		TON_historyCurrent.IN := FALSE;
	END_IF;
	TON_historyCurrent();

	// soc history
	TON_historySoc.PT := socHistoryInverval;
	TON_historySoc.IN := TRUE;
	IF TON_historySoc.Q THEN
		FOR i := 999 TO 1 BY -1 DO
			gAMS.data.history.actSoc[i] := gAMS.data.history.actSoc[i-1];
		END_FOR;
		gAMS.data.history.actSoc[0] := gAMS.data.stateOfCharge;
		TON_historySoc.IN := FALSE;
	END_IF;
	TON_historySoc();

	// voltage history
	TON_historyVoltage.PT := voltageHistoryInverval;
	TON_historyVoltage.IN := TRUE;
	IF TON_historyVoltage.Q THEN
		FOR i := 999 TO 1 BY -1 DO
			gAMS.data.history.actVoltage[i] := gAMS.data.history.actVoltage[i-1];
		END_FOR;
		gAMS.data.history.actVoltage[0] := gShunt.data.actVoltage;
		TON_historyVoltage.IN := FALSE;
	END_IF;
	TON_historyVoltage();

END_ACTION
```

#### states.st
```iecst
ACTION states:
	// Generate command ID for AMS
	IF gAMS.cmd.abort THEN
		//Signal the AMS to shutdown TS, SC and go to state idle
		gORION.state := ABORT;

		gEventLog.newEventString := 'Abort command send to AMS';
		logEvent;
	END_IF;

	// States of ORION BMS
	CASE gORION.state OF
		IDLE:
			gAMS.status.amsStateName := 'IDLE';
			gORION.relays.sdcEnable := FALSE;
			gORION.relays.precharge	:= FALSE;
			gORION.relays.airPlus	:= FALSE;
			gORION.relays.airMinus	:= FALSE;

			IF gAMS.cmd.enableSC THEN
				gAMS.cmd.enableSC := FALSE;
				gORION.state := ENABLING_SC;

				gEventLog.newEventString := 'Enable SC command send to AMS';
				logEvent;
			END_IF

		ENABLING_SC:
			gAMS.status.amsStateName := 'ENABLING_SC';

			// Settting Relays
			gORION.relays.sdcEnable := TRUE;
			gORION.relays.precharge	:= FALSE;
			gORION.relays.airPlus	:= FALSE;
			gORION.relays.airMinus	:= FALSE;

			IF gORION.status.sdcEnabled THEN
	  			gORION.state := SC_ENABLED;
			END_IF;

		SC_ENABLED:
			gAMS.status.amsStateName := 'SC_ENABLED';
			gORION.relays.sdcEnable := TRUE;
			gORION.relays.precharge	:= FALSE;
			gORION.relays.airPlus	:= FALSE;
			gORION.relays.airMinus	:= FALSE;

			IF gAMS.cmd.startPrecharge THEN
				gAMS.cmd.startPrecharge := FALSE;

				inrushCurrentDetected 	:= FALSE;
				gORION.state 			:= PRECHARGING;

				gEventLog.newEventString := 'Precharge command send to AMS';
				logEvent;
			END_IF

		PRECHARGING:
			gAMS.status.amsStateName := 'PRECHARGING';
			gORION.relays.sdcEnable := TRUE;
			gORION.relays.precharge	:= TRUE;
			gORION.relays.airPlus	:= FALSE;
			gORION.relays.airMinus	:= TRUE;

			IF gShunt.status.ok THEN
				prechargeCalculationShunt;
			ELSE
				prechargeCalculationOrion;
			END_IF;

			IF inrushCurrentDetected AND prechargeLevelReached THEN
	  			gORION.state := PRECHARGING_DONE;
			END_IF;

		PRECHARGING_DONE:
			gAMS.status.amsStateName := 'PRECHARGING_DONE';
			gORION.relays.sdcEnable := TRUE;
			gORION.relays.precharge	:= TRUE;
			gORION.relays.airPlus	:= FALSE;
			gORION.relays.airMinus	:= TRUE;

			// Set global message for general StatemMachine to continue
			gAMS.status.prechargingDone := TRUE;

			IF gAMS.cmd.enterDrive THEN
				gAMS.cmd.enterDrive 	:= FALSE;
				// Setting 500ms delay for switching off Precharge
				TON_prechargeDisableDrive.PT := T#500ms;
				TON_prechargeDisableDrive.IN := TRUE;
				gORION.state := DRIVE_PRECHARGE_ACTIVE;

				gEventLog.newEventString := 'Drive command send to AMS';
				logEvent;
			END_IF

		DRIVE_PRECHARGE_ACTIVE:
			gAMS.status.amsStateName := 'DRIVE_PRECHARGE_ACTIVE';

			gORION.relays.sdcEnable := TRUE;
			gORION.relays.precharge	:= TRUE;
			gORION.relays.airPlus	:= TRUE;
			gORION.relays.airMinus	:= TRUE;

			// Some time before disabling precharge relay
			IF TON_prechargeDisableDrive.Q THEN
				TON_prechargeDisableDrive.IN := FALSE;
				gORION.state := DRIVE;
			END_IF;

		DRIVE:
			gAMS.status.amsStateName := 'DRIVE';
			// IN drive Precharge relay should be shut off
			gORION.relays.sdcEnable := TRUE;
			gORION.relays.precharge	:= FALSE;
			gORION.relays.airPlus	:= TRUE;
			gORION.relays.airMinus	:= TRUE;

		ABORT:
			gAMS.status.amsStateName := 'ABORT';
			// state reached, Resetting command
			gAMS.cmd.abort := FALSE;
			// All relays should be shut off, to make sure no HV is on the car
			gORION.relays.sdcEnable := FALSE;
			gORION.relays.precharge	:= FALSE;
			gORION.relays.airPlus	:= FALSE;
			gORION.relays.airMinus	:= FALSE;

			// TODO: FIgure out how to know if it is safe to go to idle again
			IF gORION.data.chargeCurrent = 0 AND gSafetyChain.status.scOK_notEnabled THEN
	  			gORION.state := IDLE;
			END_IF;

		ELSE
			// IF state is outside defined states, shut off relays
			gORION.relays.sdcEnable := FALSE;
			gORION.relays.precharge	:= FALSE;
			gORION.relays.airPlus	:= FALSE;
			gORION.relays.airMinus	:= FALSE;
	END_CASE;

	// Lookup name of AMS state (Only important states)
//	CASE gAMS.status.amsState OF
//		AMS_STATE_NONE: 		gAMS.status.amsStateName := 'NONE';
//		AMS_STATE_INIT: 		gAMS.status.amsStateName := 'INIT';
//		AMS_STATE_IDLE: 		gAMS.status.amsStateName := 'IDLE';
//		AMS_STATE_ERROR: 		gAMS.status.amsStateName := 'ERROR';
//		AMS_STATE_SC_ENABLED: 	gAMS.status.amsStateName := 'SC_ENABLED';
//		AMS_STATE_TC_ENABLED: 	gAMS.status.amsStateName := 'TS_ACTIVE';
//		AMS_STATE_DRIVE: 		gAMS.status.amsStateName := 'DRIVE';
//		ELSE
//	END_CASE;

	TON_prechargeDisableDrive();

END_ACTION
```

#### prechargeCalculation.st
```iecst
ACTION prechargeCalculationOrion:

	// Check if any inrush current, to make sure precharging is acutally being performed
	IF gORION.data.outputCurrent > 0 THEN
		inrushCurrentDetected := TRUE;
	END_IF;

	// Calculate the voltage on the voltage on the Car side based on precharge resistor and pack voltage
	gORION.data.carVoltage := gORION.data.packVoltage - ABS(prechargeResistance * gORION.data.chargeCurrent);
	gORION.data.prechargeLevel := gORION.data.packVoltage / gORION.data.carVoltage;

	IF gORION.data.prechargeLevel >= requiredPrechargeLevel AND gORION.data.outputCurrent = 0 THEN
		prechargeLevelReached := TRUE;
	ELSE
		prechargeLevelReached := FALSE;
	END_IF;

END_ACTION

ACTION prechargeCalculationShunt:

	IF gORION.data.packVoltage > 0 THEN
		IF gShunt.data.actVoltage >= gORION.data.packVoltage * requiredPrechargeLevel THEN
			prechargeLevelReached := TRUE;
		ELSE
			prechargeLevelReached := FALSE;
		END_IF;
	ELSE
		prechargeLevelReached := FALSE;
	END_IF

END_ACTION
```

#### errors.st
```iecst
ACTION errorsInit_action:
	// Set a timeout period and start all error timers
	FOR i := 0 TO 21 DO
		gAMS.status.error.errorTimers[i](IN := TRUE, PT := T#100ms);
	END_FOR;

	// Init all errors as inactive
	gAMS.status.error.lowVoltage 			:= FALSE;
	gAMS.status.error.highVoltage 			:= FALSE;
	gAMS.status.error.lowTemp 				:= FALSE;
	gAMS.status.error.highTemp 				:= FALSE;
	gAMS.status.error.ltc6813Com 			:= FALSE;
	gAMS.status.error.shuntCom 				:= FALSE;
	gAMS.status.error.openSc 				:= FALSE;
	gAMS.status.error.closeSc 				:= FALSE;
	gAMS.status.error.openAirMinus 			:= FALSE;
	gAMS.status.error.closeAirMinus 		:= FALSE;
	gAMS.status.error.openAirPlus 			:= FALSE;
	gAMS.status.error.closeAirPlus 			:= FALSE;
	gAMS.status.error.openPrePlus 			:= FALSE;
	gAMS.status.error.closePrePlus  		:= FALSE;
	gAMS.status.error.preTimeout 			:= FALSE;
	gAMS.status.error.unexpectedChargeRate 	:= FALSE;
	gAMS.status.error.bankCountMismatch 	:= FALSE;
	gAMS.status.error.unexpectedTsCurrent 	:= FALSE;
	gAMS.status.error.relayFailed 			:= FALSE;
	gAMS.status.error.scBroken 				:= FALSE;
	gAMS.status.error.unfitChargeVoltage 	:= FALSE;
	gAMS.status.error.monitorError 			:= FALSE;
END_ACTION

ACTION error_action:
	// Service all error timers
	FOR i := 0 TO 21 DO
		gAMS.status.error.errorTimers[i]();
	END_FOR;

	(*  Write timer state to error flag. If timer runs out that means the error is inactive.
		The check should only run when the node is not in state INIT which also gives the timeout timers time to run out to begin with
		so no premature errors will be reported.*)

	//	1 ERROR_AMS_CELL_VOLTAGE_LOW
	//	2 ERROR_AMS_CELL_VOLTAGE_HIGH
	//	3 ERROR_AMS_CELL_TEMP_LOW
	//	4 ERROR_AMS_CELL_TEMP_HIGH
	//	5 ERROR_AMS_LTC6813_COMM
	//	6 ERROR_AMS_SHUNT_COMM
	//	7 ERROR_AMS_UNABLE_TO_OPEN_SC
	//	8 ERROR_AMS_UNABLE_TO_CLOSE_SC
	//	9 ERROR_AMS_UNABLE_TO_OPEN_AIR-
	//	10 ERROR_AMS_UNABLE_TO_CLOSE_AIR-
	//	11 ERROR_AMS_UNABLE_TO_OPEN_AIR+
	//	12 ERROR_AMS_UNABLE_TO_CLOSE_AIR+
	//	13 ERROR_AMS_UNABLE_TO_OPEN_PRE+
	//	14 ERROR_AMS_UNABLE_TO_CLOSE_PRE+
	//	15 ERROR_AMS_PRE_TIMEOUT
	//	16 ERROR_AMS_UNEXPECTED_CHARGE_RATE
	//	17 ERROR_AMS_BANK_COUNT_MISMATCH
	//	18 ERROR_AMS_UNEXSPECPTED_TS_CURRENT
	//	19 ERROR_AMS_RELAY_FAIELD
	//	20 ERROR_AMS_SC_BROKEN
	//	21 AMS_UNFIT_CHARGE_VOLTAGE
	//	22 AMS_MONITOR_ERROR
	IF gStateMachine.status.state <> STATE_INITIALIZE THEN
		gAMS.status.error.lowVoltage 			:= NOT gAMS.status.error.errorTimers[0].Q;
		gAMS.status.error.highVoltage 			:= NOT gAMS.status.error.errorTimers[1].Q;
		gAMS.status.error.lowTemp 				:= NOT gAMS.status.error.errorTimers[2].Q;
		gAMS.status.error.highTemp 				:= NOT gAMS.status.error.errorTimers[3].Q;
		gAMS.status.error.ltc6813Com 			:= NOT gAMS.status.error.errorTimers[4].Q;
		gAMS.status.error.shuntCom 				:= NOT gAMS.status.error.errorTimers[5].Q;
		gAMS.status.error.openSc 				:= NOT gAMS.status.error.errorTimers[6].Q;
		gAMS.status.error.closeSc 				:= NOT gAMS.status.error.errorTimers[7].Q;
		gAMS.status.error.openAirMinus 			:= NOT gAMS.status.error.errorTimers[8].Q;
		gAMS.status.error.closeAirMinus 		:= NOT gAMS.status.error.errorTimers[9].Q;
		gAMS.status.error.openAirPlus 			:= NOT gAMS.status.error.errorTimers[10].Q;
		gAMS.status.error.closeAirPlus 			:= NOT gAMS.status.error.errorTimers[11].Q;
		gAMS.status.error.openPrePlus 			:= NOT gAMS.status.error.errorTimers[12].Q;
		gAMS.status.error.closePrePlus  		:= NOT gAMS.status.error.errorTimers[13].Q;
		gAMS.status.error.preTimeout 			:= NOT gAMS.status.error.errorTimers[14].Q;
		gAMS.status.error.unexpectedChargeRate 	:= NOT gAMS.status.error.errorTimers[15].Q;
		gAMS.status.error.bankCountMismatch 	:= NOT gAMS.status.error.errorTimers[16].Q;
		gAMS.status.error.unexpectedTsCurrent 	:= NOT gAMS.status.error.errorTimers[17].Q;
		gAMS.status.error.relayFailed 			:= NOT gAMS.status.error.errorTimers[18].Q;
		gAMS.status.error.scBroken 				:= NOT gAMS.status.error.errorTimers[19].Q;
		gAMS.status.error.unfitChargeVoltage 	:= NOT gAMS.status.error.errorTimers[20].Q;
		gAMS.status.error.monitorError 			:= NOT gAMS.status.error.errorTimers[21].Q;
	END_IF;

	gAMS.status.hasError := gAMS.status.error.lowVoltage 		 OR gAMS.status.error.highVoltage 			OR
							gAMS.status.error.lowTemp 			 OR gAMS.status.error.highTemp 				OR
							gAMS.status.error.ltc6813Com 		 OR gAMS.status.error.shuntCom 				OR
							gAMS.status.error.openSc 			 OR gAMS.status.error.closeSc 				OR
							gAMS.status.error.openAirMinus 	 	 OR gAMS.status.error.closeAirMinus 		OR
							gAMS.status.error.openAirPlus 	 	 OR gAMS.status.error.closeAirPlus 			OR
							gAMS.status.error.openPrePlus 	 	 OR gAMS.status.error.closePrePlus 			OR
							gAMS.status.error.preTimeout 		 OR gAMS.status.error.unexpectedChargeRate 	OR
							gAMS.status.error.bankCountMismatch  OR gAMS.status.error.unexpectedTsCurrent 	OR
							gAMS.status.error.relayFailed 		 OR gAMS.status.error.scBroken 				OR
							gAMS.status.error.unfitChargeVoltage OR gAMS.status.error.monitorError;
END_ACTION
```

#### orionErrorAction.st
```iecst
ACTION orionErrorAction:

	// If charger intends to do an AMS error, force an abort:
	IF NOT gAMS.status.relayState.dischargeRelayEnabled THEN
		gAMS.cmd.abort;
		gAMS.status.errorInfo := 'DischargeEnable pin is FALSE';
	END_IF;

	// If voltage too high force an abort
	IF gAMS.status.error.lowVoltage THEN
		gAMS.cmd.abort;
		gAMS.status.errorInfo := 'Voltage of a cell is too low';
	END_IF;

	// If Temp is too high
	IF gAMS.status.error.highTemp THEN
		gAMS.cmd.abort;
		gAMS.status.errorInfo := 'Temperature of a cell is too high';
	END_IF;

	// Manual check of  cell temp
	IF gAMS.data.cellTempMax > 60 THEN
		gAMS.cmd.abort;
		gAMS.status.errorInfo := 'Temperature of a cell is above 60 Degree';
	END_IF;

	// charge is above Discharge Current Limit (DCL)
	IF gORION.data.outputCurrent > gORION.data.DCL THEN
		gAMS.cmd.abort;
		gAMS.status.errorInfo := 'Charge Current Limit(CCL) exceeded';
	END_IF;

	// Rolling counter has changed
	IF gORION.data.rollingCounter <> gORION.data.rollingCounterOld THEN
		gORION.data.TON_counter.IN := FALSE;
		gORION.data.TON_counter();
		gORION.data.TON_counter.IN := TRUE;
	END_IF;
	gORION.data.rollingCounterOld := gORION.data.rollingCounter;

	// Timeout on the rolling counter
	IF gORION.data.TON_counter.Q THEN
		gAMS.cmd.abort := TRUE;
		gAMS.status.error.amsError 	:= TRUE;
		gORION.status.commTimeout	:= TRUE;
		gAMS.status.errorInfo := 'Timeout of commnication with ORION BMS';
	ELSE
		gORION.status.commTimeout	:= FALSE;
	END_IF;

	gORION.data.TON_counter();

END_ACTION
```

### Program Logical/AMS_and_Shunt/CAN/AMS_CAN (IEC)

#### Variables.var - Local variables
```iecst
VAR
	dataArr : ARRAY[0..3] OF BYTE;
	data : UDINT;
	ArCanSend_0 : ArCanSend;
	CCL_KW_Temp : INT;
	DCL_KW_Temp : INT;
	ArCanReceive_0 : ArCanReceive;
	ArCanSetBaudrate_0 : ArCanSetBaudrate;
	communicationState : CAN_STATES;
	deviceName : STRING[127];
	i : USINT;
	TON_sendTimer : TON;
	TON_shuntDisconnected : TON;
	TON_amsDisconnected : TON;
	TX_CAN_ID_BASE : {REDUND_UNREPLICABLE} UDINT := 0;
	SHUNT_ID_BASE : {REDUND_UNREPLICABLE} UDINT := 0;
	RX_ORION_ID_BASE : {REDUND_UNREPLICABLE} UDINT := 0;
	TX_ORION_ID_BASE : {REDUND_UNREPLICABLE} UDINT := 0;
	RX_CAN_ID_BASE : {REDUND_UNREPLICABLE} UDINT := 0;
	NO_OF_BANKS : USINT := 0;
	frameId : UDINT;
	errorId : USINT;
	bankId : USINT;
	groupId : USINT;
	messageCounterRec : USINT;
	messageCounterSent : USINT;
	messageCounter : USINT;
	cellId : USINT := 0;
	checksumCalculated : UDINT;
	checksumGiven : USINT;
	checksumValidate : USINT;
	tempVoltageLow : USINT;
	tempVoltageHigh : USINT;
	tempVoltage : UINT;
	packCurrent : INT;
	packVoltage : UINT;
	packPower : INT;
	checksumCorrect : USINT;
	mpeTemp : USINT;
	mpo1Temp : USINT;
	mpo2Temp : USINT;
	mpo3Temp : USINT;
	mpoTemp : USINT;
	bankCellId : USINT;
	j : USINT;
END_VAR
```

#### AMS_Send.st
```iecst
ACTION AMS_Send:

	(* Set timer *)
	TON_sendTimer.PT := T#50ms;

	(* If timer runs out *)
	IF TON_sendTimer.Q THEN
		IF ArCanSend_0.NumberOfFreeBuffers > 1010 THEN
			// msg_x05; // Should be used with the old AMS
			FOR i:=0 TO 2-1 DO // Number of messages minus 1
				messageCounterSent := messageCounterSent + 1;
				CASE i OF
					0:
						msg_orion_tx20;
					1:
						msg_orion_tx21;
				END_CASE;
			END_FOR;
		END_IF;

		(* Reset timer *)
		TON_sendTimer(IN:=FALSE);
	END_IF

	(* Start timer *)
	TON_sendTimer(IN:=TRUE);

END_ACTION
```

#### ams_tx_msgs.st
```iecst
ACTION msg_x05:

	// Command ID
	ArCanSend_0.Frame.Data[0].0 := gAMS.cmd.commandId.0;
	ArCanSend_0.Frame.Data[0].1 := gAMS.cmd.commandId.1;
	ArCanSend_0.Frame.Data[0].2 := gAMS.cmd.commandId.2;
	ArCanSend_0.Frame.Data[0].3 := gAMS.cmd.commandId.3;

	// Bank count
	ArCanSend_0.Frame.Data[0].4 := gAMS.cmd.bankCount.0;
	ArCanSend_0.Frame.Data[0].5 := gAMS.cmd.bankCount.1;
	ArCanSend_0.Frame.Data[0].6 := gAMS.cmd.bankCount.2;
	ArCanSend_0.Frame.Data[0].7 := gAMS.cmd.bankCount.3;

	// Message counter
	memcpy(ADR(ArCanSend_0.Frame.Data[1]), ADR(messageCounter), 1);

	IF NOT gIsSimulation THEN
		(* Set ID *)
		ArCanSend_0.Frame.ID 			:= TX_CAN_ID_BASE + 16#005;

		(* Set DLC *)
		ArCanSend_0.Frame.DataLength 	:= 2;

		(* Send message *)
		ArCanSend_0(SendFrame := TRUE);
		ArCanSend_0(SendFrame := FALSE);
	END_IF;

	// Increment message counter
	messageCounter := messageCounter + 1;
END_ACTION
```

#### orion_tx_msgs.st
```iecst
ACTION msg_orion_tx20:

	// Command for enabling and disabling MPE = Sdc_en
	gAMS.cmd.mpe.0 := gORION.relays.sdcEnable;
	memcpy(ADR(ArCanSend_0.Frame.Data[0]), ADR(gAMS.cmd.mpe), 1);

	// Message counter
	// memcpy(ADR(ArCanSend_0.Frame.Data[1]), ADR(messageCounter), 1);

	IF NOT gIsSimulation THEN
		(* Set ID *)
		ArCanSend_0.Frame.ID 			:= TX_ORION_ID_BASE + 16#020;

		(* Set DLC *)
		ArCanSend_0.Frame.DataLength 	:= 8;

		(* Send message *)
		ArCanSend_0(SendFrame := TRUE);
		ArCanSend_0(SendFrame := FALSE);
	END_IF;

	// Increment message counter
	messageCounter := messageCounter + 1;
END_ACTION

ACTION msg_orion_tx21:

	// Command ID
	// MPO1 - Precharge relay state
	gAMS.cmd.mpo1.0 := gORION.relays.precharge;
	memcpy(ADR(ArCanSend_0.Frame.Data[0]), ADR(gAMS.cmd.mpo1), 1);
	// MPO2 - AIR+ relay state
	gAMS.cmd.mpo2.0 := gORION.relays.airPlus;
	memcpy(ADR(ArCanSend_0.Frame.Data[1]), ADR(gAMS.cmd.mpo2), 1);
	// MPO3 - AIR- relay state
	gAMS.cmd.mpo3.0 := gORION.relays.airMinus;
	memcpy(ADR(ArCanSend_0.Frame.Data[2]), ADR(gAMS.cmd.mpo3), 1);

	// Message counter
	// memcpy(ADR(ArCanSend_0.Frame.Data[1]), ADR(messageCounter), 1);

	IF NOT gIsSimulation THEN
		(* Set ID *)
		ArCanSend_0.Frame.ID 			:= TX_ORION_ID_BASE + 16#021;

		(* Set DLC *)
		ArCanSend_0.Frame.DataLength 	:= 8;

		(* Send message *)
		ArCanSend_0(SendFrame := TRUE);
		ArCanSend_0(SendFrame := FALSE);
	END_IF;

	// Increment message counter
	messageCounter := messageCounter + 1;
END_ACTION
```

#### functions.st
```iecst
ACTION getBankIdAndGroupId:
	// Bank ID
	bankId.2 := ArCanReceive_0.ReceivedFrame.Data[0].7;
	bankId.1 := ArCanReceive_0.ReceivedFrame.Data[0].6;
	bankId.0 := ArCanReceive_0.ReceivedFrame.Data[0].5;
	bankId := bankId - 1;

	// Group ID
	groupId.2 := ArCanReceive_0.ReceivedFrame.Data[0].2;
	groupId.1 := ArCanReceive_0.ReceivedFrame.Data[0].1;
	groupId.0 := ArCanReceive_0.ReceivedFrame.Data[0].0;
END_ACTION

ACTION cellidToBankAndCell:
	// COnverting the send cell id from the orion BMS to Bank and specific cell
	bankId := 0;
	bankCellId := cellId;
	FOR i := 0 TO BANK_COUNT - 1 DO
		IF bankCellId >= 36 THEN
			bankCellId := bankCellId - 36;
			bankId := bankId + 1;
		ELSE
			EXIT;
		END_IF;
	END_FOR;

END_ACTION

ACTION appendTemps:

	FOR i:=0 TO (SIZEOF(gAMS.status.bank)/SIZEOF(gAMS.status.bank[0]))-1 DO
		FOR j := 0 TO (SIZEOF(gAMS.status.bank[0].temperatures)/SIZEOF(gAMS.status.bank[0].temperatures[0]))-1 DO
			gAMS.status.bank[i].temperatures[j] := gAMS.data.cellTempMax;
		END_FOR;
	END_FOR;
END_ACTION
```

#### Program Logical/AMS_and_Shunt/CAN/AMS_CAN/Receive/Messages
